Yaskawa INFORM job: DEMO_ROOF_SIDE_0625_3PAINT_4.JBI

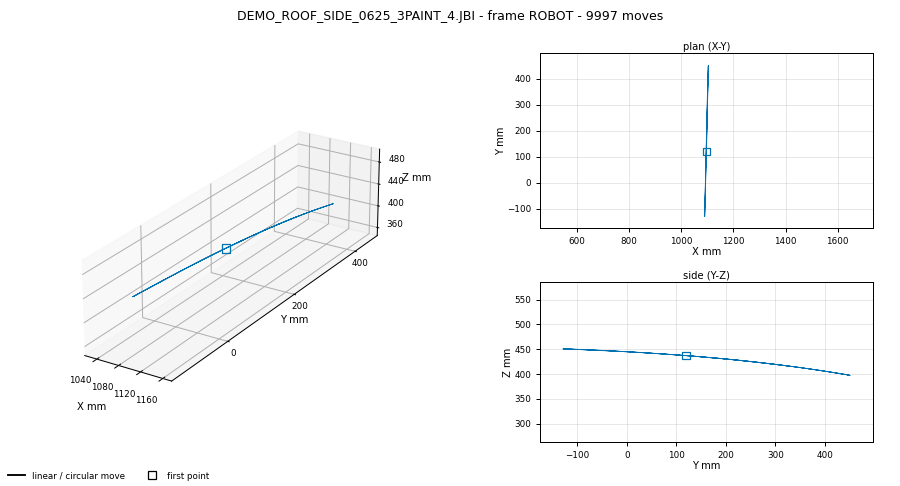
[picture p0: tool path of DEMO_ROOF_SIDE_0625_3PAINT_4.JBI in frame ROBOT, 9997 of 9997 moves have a stored position in this frame; points joined in program order, loops and branches not executed]
/JOB
//NAME DEMO_ROOF_SIDE_0625_3PAINT4
//POS
///NPOS 9997,0,0,0,0,0
///TOOL 0
///USER 0
///POSTYPE ROBOT
///RECTAN
///RCONF 1,0,0,0,0,0,0,0,0,0,0,0,0,0,0,0,0,0,0,0,0,0,0,0
C00000=1096.596,120.158,437.402,176.522,16.758,152.268
C00001=1096.602,120.407,437.382,176.524,16.758,152.268
C00002=1096.608,120.656,437.363,176.527,16.758,152.267
C00003=1096.614,120.905,437.344,176.530,16.759,152.267
C00004=1096.619,121.154,437.325,176.533,16.759,152.267
C00005=1096.625,121.404,437.306,176.536,16.760,152.266
C00006=1096.630,121.653,437.287,176.539,16.761,152.266
C00007=1096.636,121.902,437.267,176.541,16.761,152.265
C00008=1096.641,122.152,437.247,176.544,16.762,152.265
C00009=1096.646,122.400,437.228,176.546,16.761,152.264
C00010=1096.652,122.650,437.209,176.549,16.762,152.264
C00011=1096.658,122.899,437.189,176.552,16.763,152.263
C00012=1096.664,123.148,437.170,176.555,16.763,152.263
C00013=1096.669,123.397,437.150,176.558,16.764,152.262
C00014=1096.675,123.647,437.131,176.561,16.764,152.262
C00015=1096.681,123.896,437.111,176.563,16.765,152.262
C00016=1096.686,124.144,437.092,176.566,16.765,152.261
C00017=1096.692,124.394,437.073,176.569,16.766,152.261
C00018=1096.697,124.643,437.054,176.571,16.766,152.260
C00019=1096.703,124.892,437.034,176.575,16.766,152.260
C00020=1096.709,125.141,437.015,176.578,16.767,152.259
C00021=1096.715,125.391,436.995,176.580,16.767,152.259
C00022=1096.720,125.640,436.975,176.583,16.768,152.258
C00023=1096.726,125.889,436.955,176.585,16.768,152.258
C00024=1096.731,126.138,436.936,176.589,16.768,152.257
C00025=1096.737,126.387,436.917,176.592,16.769,152.257
C00026=1096.743,126.636,436.897,176.594,16.769,152.256
C00027=1096.749,126.885,436.877,176.597,16.770,152.256
C00028=1096.754,127.135,436.858,176.600,16.770,152.256
C00029=1096.760,127.383,436.838,176.602,16.770,152.255
C00030=1096.766,127.659,436.817,176.606,16.771,152.254
C00031=1096.773,127.934,436.795,176.609,16.771,152.254
C00032=1096.779,128.209,436.774,176.612,16.772,152.253
C00033=1096.785,128.484,436.751,176.615,16.772,152.253
C00034=1096.791,128.733,436.731,176.618,16.773,152.252
C00035=1096.796,128.982,436.712,176.621,16.773,152.252
C00036=1096.802,129.231,436.693,176.624,16.773,152.251
C00037=1096.808,129.480,436.673,176.627,16.774,152.251
C00038=1096.814,129.729,436.653,176.629,16.774,152.250
C00039=1096.819,129.979,436.634,176.632,16.774,152.250
C00040=1096.825,130.227,436.614,176.636,16.775,152.249
C00041=1096.830,130.477,436.594,176.638,16.775,152.249
C00042=1096.836,130.726,436.574,176.641,16.775,152.248
C00043=1096.842,130.975,436.555,176.644,16.776,152.248
C00044=1096.848,131.225,436.535,176.646,16.776,152.247
C00045=1096.854,131.474,436.514,176.649,16.777,152.247
C00046=1096.859,131.723,436.495,176.653,16.777,152.246
C00047=1096.865,131.972,436.475,176.655,16.777,152.246
C00048=1096.871,132.221,436.456,176.658,16.778,152.245
C00049=1096.876,132.470,436.435,176.661,16.778,152.245
C00050=1096.882,132.719,436.415,176.664,16.778,152.244
C00051=1096.888,132.969,436.396,176.667,16.778,152.244
C00052=1096.893,133.218,436.376,176.670,16.779,152.243
C00053=1096.899,133.467,436.356,176.672,16.779,152.243
C00054=1096.904,133.716,436.336,176.676,16.779,152.242
C00055=1096.910,133.965,436.316,176.679,16.780,152.242
C00056=1096.916,134.214,436.296,176.681,16.780,152.241
C00057=1096.921,134.464,436.276,176.684,16.781,152.241
C00058=1096.927,134.713,436.256,176.687,16.781,152.240
C00059=1096.932,134.962,436.235,176.690,16.781,152.240
C00060=1096.938,135.211,436.216,176.693,16.782,152.239
C00061=1096.944,135.460,436.196,176.696,16.782,152.239
C00062=1096.949,135.709,436.176,176.698,16.782,152.238
C00063=1096.955,135.958,436.156,176.701,16.783,152.238
C00064=1096.961,136.207,436.135,176.705,16.783,152.237
C00065=1096.966,136.456,436.116,176.707,16.783,152.237
C00066=1096.972,136.706,436.095,176.710,16.784,152.236
C00067=1096.978,136.954,436.075,176.713,16.784,152.236
C00068=1096.983,137.204,436.055,176.716,16.785,152.235
C00069=1096.989,137.452,436.035,176.719,16.785,152.235
C00070=1096.994,137.702,436.016,176.722,16.785,152.234
C00071=1097.000,137.951,435.995,176.725,16.785,152.234
C00072=1097.006,138.200,435.975,176.727,16.785,152.233
C00073=1097.012,138.450,435.954,176.731,16.786,152.233
C00074=1097.018,138.698,435.934,176.734,16.786,152.232
C00075=1097.023,138.947,435.914,176.736,16.786,152.232
C00076=1097.029,139.196,435.894,176.739,16.787,152.231
C00077=1097.034,139.446,435.874,176.743,16.787,152.231
C00078=1097.039,139.695,435.853,176.745,16.787,152.230
C00079=1097.045,139.944,435.833,176.748,16.788,152.230
C00080=1097.050,140.193,435.813,176.751,16.788,152.229
C00081=1097.056,140.442,435.793,176.755,16.788,152.228
C00082=1097.062,140.692,435.772,176.757,16.788,152.228
C00083=1097.068,140.941,435.752,176.760,16.789,152.227
C00084=1097.073,141.190,435.731,176.763,16.789,152.227
C00085=1097.079,141.439,435.711,176.766,16.789,152.226
C00086=1097.085,141.688,435.691,176.769,16.790,152.226
C00087=1097.090,141.937,435.670,176.772,16.790,152.225
C00088=1097.095,142.186,435.650,176.775,16.790,152.225
C00089=1097.101,142.435,435.630,176.778,16.790,152.224
C00090=1097.107,142.684,435.609,176.781,16.791,152.224
C00091=1097.112,142.934,435.588,176.784,16.791,152.223
C00092=1097.118,143.182,435.568,176.786,16.791,152.223
C00093=1097.124,143.432,435.548,176.790,16.792,152.222
C00094=1097.130,143.707,435.525,176.793,16.792,152.222
C00095=1097.136,143.981,435.503,176.797,16.792,152.221
C00096=1097.142,144.256,435.480,176.800,16.792,152.220
C00097=1097.149,144.530,435.458,176.803,16.793,152.220
C00098=1097.154,144.780,435.437,176.806,16.793,152.219
C00099=1097.160,145.029,435.416,176.809,16.793,152.219
C00100=1097.165,145.278,435.396,176.812,16.793,152.218
C00101=1097.171,145.527,435.376,176.815,16.794,152.218
C00102=1097.176,145.776,435.355,176.817,16.794,152.217
C00103=1097.182,146.025,435.333,176.821,16.794,152.216
C00104=1097.188,146.274,435.314,176.824,16.795,152.216
C00105=1097.194,146.523,435.293,176.827,16.795,152.215
C00106=1097.199,146.772,435.272,176.830,16.795,152.215
C00107=1097.205,147.022,435.251,176.833,16.795,152.214
C00108=1097.211,147.270,435.231,176.836,16.795,152.214
C00109=1097.216,147.519,435.210,176.839,16.795,152.213
C00110=1097.222,147.769,435.190,176.842,16.796,152.213
C00111=1097.227,148.018,435.169,176.845,16.796,152.212
C00112=1097.234,148.267,435.148,176.848,16.796,152.211
C00113=1097.239,148.516,435.128,176.851,16.796,152.211
C00114=1097.244,148.765,435.107,176.854,16.796,152.210
C00115=1097.250,149.015,435.086,176.857,16.797,152.210
C00116=1097.256,149.263,435.065,176.861,16.797,152.209
C00117=1097.261,149.512,435.044,176.863,16.797,152.209
C00118=1097.266,149.761,435.024,176.866,16.797,152.208
C00119=1097.273,150.010,435.003,176.870,16.798,152.207
C00120=1097.278,150.259,434.982,176.872,16.797,152.207
C00121=1097.284,150.509,434.962,176.875,16.798,152.206
C00122=1097.289,150.757,434.940,176.879,16.798,152.206
C00123=1097.295,151.007,434.919,176.882,16.799,152.205
C00124=1097.301,151.255,434.898,176.884,16.798,152.205
C00125=1097.306,151.505,434.878,176.888,16.799,152.204
C00126=1097.312,151.754,434.857,176.891,16.799,152.203
C00127=1097.317,152.003,434.835,176.894,16.799,152.203
C00128=1097.322,152.252,434.815,176.897,16.799,152.202
C00129=1097.329,152.501,434.793,176.900,16.800,152.202
C00130=1097.334,152.750,434.773,176.903,16.800,152.201
C00131=1097.339,152.999,434.751,176.906,16.800,152.201
C00132=1097.345,153.248,434.731,176.909,16.800,152.200
C00133=1097.351,153.497,434.710,176.912,16.801,152.200
C00134=1097.357,153.746,434.689,176.915,16.801,152.199
C00135=1097.362,153.995,434.669,176.918,16.800,152.198
C00136=1097.368,154.244,434.647,176.921,16.801,152.198
C00137=1097.374,154.493,434.626,176.925,16.801,152.197
C00138=1097.380,154.743,434.605,176.928,16.801,152.197
C00139=1097.385,154.991,434.584,176.930,16.801,152.196
C00140=1097.391,155.240,434.563,176.934,16.801,152.195
C00141=1097.397,155.489,434.541,176.937,16.802,152.195
C00142=1097.402,155.739,434.521,176.940,16.802,152.194
C00143=1097.407,155.987,434.499,176.943,16.802,152.194
C00144=1097.413,156.237,434.478,176.946,16.802,152.193
C00145=1097.418,156.486,434.457,176.949,16.802,152.192
C00146=1097.424,156.735,434.435,176.953,16.803,152.192
C00147=1097.430,156.984,434.415,176.955,16.802,152.191
C00148=1097.435,157.233,434.393,176.958,16.803,152.191
C00149=1097.441,157.482,434.372,176.962,16.803,152.190
C00150=1097.447,157.731,434.351,176.965,16.803,152.190
C00151=1097.452,157.979,434.330,176.968,16.803,152.189
C00152=1097.458,158.229,434.308,176.971,16.803,152.188
C00153=1097.463,158.478,434.287,176.974,16.804,152.188
C00154=1097.469,158.727,434.265,176.978,16.804,152.187
C00155=1097.475,158.976,434.244,176.980,16.803,152.187
C00156=1097.480,159.226,434.223,176.983,16.804,152.186
C00157=1097.486,159.474,434.202,176.987,16.804,152.185
C00158=1097.493,159.748,434.178,176.990,16.804,152.185
C00159=1097.499,160.023,434.155,176.994,16.804,152.184
C00160=1097.505,160.298,434.132,176.997,16.804,152.183
C00161=1097.510,160.572,434.107,177.001,16.804,152.183
C00162=1097.517,160.822,434.086,177.004,16.805,152.182
C00163=1097.522,161.070,434.064,177.007,16.805,152.181
C00164=1097.528,161.320,434.044,177.010,16.804,152.181
C00165=1097.533,161.568,434.022,177.013,16.805,152.180
C00166=1097.538,161.817,434.000,177.016,16.805,152.180
C00167=1097.544,162.066,433.979,177.020,16.805,152.179
C00168=1097.550,162.315,433.958,177.023,16.805,152.178
C00169=1097.555,162.564,433.935,177.026,16.805,152.178
C00170=1097.561,162.814,433.915,177.029,16.806,152.177
C00171=1097.566,163.063,433.893,177.032,16.806,152.177
C00172=1097.572,163.312,433.871,177.036,16.806,152.176
C00173=1097.577,163.560,433.850,177.038,16.806,152.175
C00174=1097.583,163.810,433.828,177.041,16.806,152.175
C00175=1097.588,164.058,433.806,177.045,16.806,152.174
C00176=1097.594,164.308,433.784,177.048,16.806,152.174
C00177=1097.599,164.556,433.763,177.051,16.807,152.173
C00178=1097.605,164.806,433.741,177.054,16.807,152.173
C00179=1097.610,165.054,433.719,177.057,16.807,152.172
C00180=1097.616,165.303,433.698,177.061,16.807,152.171
C00181=1097.621,165.552,433.676,177.064,16.807,152.171
C00182=1097.627,165.801,433.654,177.067,16.808,152.170
C00183=1097.632,166.050,433.632,177.070,16.807,152.169
C00184=1097.638,166.299,433.611,177.073,16.807,152.169
C00185=1097.643,166.548,433.589,177.076,16.808,152.168
C00186=1097.649,166.797,433.567,177.080,16.808,152.168
C00187=1097.654,167.046,433.545,177.083,16.808,152.167
C00188=1097.660,167.295,433.524,177.086,16.807,152.166
C00189=1097.665,167.544,433.502,177.089,16.808,152.166
C00190=1097.671,167.793,433.480,177.093,16.808,152.165
C00191=1097.676,168.042,433.458,177.096,16.808,152.164
C00192=1097.682,168.291,433.437,177.099,16.809,152.164
C00193=1097.687,168.540,433.415,177.102,16.808,152.163
C00194=1097.693,168.790,433.393,177.105,16.808,152.163
C00195=1097.698,169.038,433.371,177.109,16.809,152.162
C00196=1097.704,169.288,433.350,177.112,16.809,152.161
C00197=1097.709,169.536,433.327,177.115,16.808,152.161
C00198=1097.716,169.785,433.306,177.118,16.808,152.160
C00199=1097.721,170.034,433.283,177.121,16.809,152.159
C00200=1097.727,170.283,433.262,177.125,16.809,152.159
C00201=1097.732,170.532,433.240,177.128,16.809,152.158
C00202=1097.738,170.780,433.218,177.131,16.808,152.158
C00203=1097.743,171.030,433.196,177.134,16.809,152.157
C00204=1097.749,171.279,433.173,177.138,16.809,152.156
C00205=1097.754,171.528,433.152,177.141,16.809,152.156
C00206=1097.760,171.777,433.129,177.144,16.809,152.155
C00207=1097.766,172.026,433.108,177.148,16.809,152.154
C00208=1097.771,172.275,433.086,177.150,16.809,152.154
C00209=1097.777,172.524,433.064,177.154,16.809,152.153
C00210=1097.782,172.772,433.042,177.157,16.809,152.152
C00211=1097.788,173.022,433.019,177.161,16.810,152.152
C00212=1097.794,173.271,432.998,177.164,16.809,152.151
C00213=1097.799,173.519,432.975,177.167,16.809,152.150
C00214=1097.805,173.768,432.953,177.170,16.809,152.150
C00215=1097.811,174.018,432.931,177.174,16.809,152.149
C00216=1097.816,174.267,432.908,177.177,16.810,152.149
C00217=1097.822,174.515,432.887,177.180,16.809,152.148
C00218=1097.827,174.765,432.865,177.183,16.809,152.147
C00219=1097.833,175.014,432.842,177.186,16.809,152.147
C00220=1097.839,175.262,432.821,177.190,16.809,152.146
C00221=1097.844,175.511,432.798,177.193,16.809,152.145
C00222=1097.851,175.785,432.774,177.197,16.809,152.144
C00223=1097.857,176.060,432.749,177.201,16.809,152.144
C00224=1097.864,176.334,432.724,177.204,16.809,152.143
C00225=1097.869,176.608,432.700,177.208,16.809,152.142
C00226=1097.875,176.857,432.677,177.211,16.809,152.142
C00227=1097.881,177.106,432.656,177.214,16.809,152.141
C00228=1097.887,177.355,432.633,177.218,16.809,152.140
C00229=1097.892,177.604,432.611,177.222,16.809,152.140
C00230=1097.898,177.852,432.589,177.224,16.809,152.139
C00231=1097.903,178.102,432.566,177.228,16.809,152.138
C00232=1097.909,178.351,432.543,177.231,16.809,152.138
C00233=1097.914,178.600,432.521,177.234,16.809,152.137
C00234=1097.920,178.848,432.499,177.238,16.809,152.136
C00235=1097.926,179.097,432.476,177.241,16.809,152.136
C00236=1097.931,179.346,432.454,177.244,16.808,152.135
C00237=1097.938,179.595,432.432,177.248,16.808,152.134
C00238=1097.943,179.845,432.409,177.251,16.809,152.134
C00239=1097.949,180.093,432.386,177.254,16.809,152.133
C00240=1097.954,180.342,432.364,177.258,16.809,152.132
C00241=1097.960,180.591,432.342,177.262,16.809,152.131
C00242=1097.966,180.840,432.319,177.264,16.808,152.131
C00243=1097.972,181.089,432.296,177.268,16.808,152.130
C00244=1097.977,181.338,432.274,177.271,16.808,152.129
C00245=1097.984,181.587,432.252,177.275,16.808,152.129
C00246=1097.989,181.836,432.229,177.278,16.808,152.128
C00247=1097.994,182.084,432.207,177.282,16.808,152.127
C00248=1098.000,182.333,432.184,177.284,16.808,152.127
C00249=1098.006,182.582,432.162,177.288,16.808,152.126
C00250=1098.012,182.831,432.139,177.291,16.808,152.125
C00251=1098.018,183.080,432.117,177.295,16.808,152.125
C00252=1098.023,183.329,432.094,177.298,16.808,152.124
C00253=1098.029,183.578,432.071,177.302,16.808,152.123
C00254=1098.036,183.827,432.048,177.305,16.807,152.123
C00255=1098.041,184.076,432.025,177.308,16.807,152.122
C00256=1098.047,184.325,432.003,177.312,16.807,152.121
C00257=1098.052,184.573,431.981,177.315,16.807,152.120
C00258=1098.058,184.822,431.958,177.319,16.807,152.120
C00259=1098.063,185.071,431.935,177.322,16.807,152.119
C00260=1098.069,185.320,431.912,177.325,16.806,152.118
C00261=1098.075,185.569,431.889,177.328,16.807,152.118
C00262=1098.080,185.818,431.866,177.332,16.807,152.117
C00263=1098.086,186.067,431.844,177.335,16.807,152.116
C00264=1098.092,186.316,431.821,177.339,16.807,152.116
C00265=1098.097,186.564,431.798,177.342,16.807,152.115
C00266=1098.102,186.813,431.775,177.346,16.807,152.114
C00267=1098.108,187.062,431.752,177.349,16.807,152.114
C00268=1098.113,187.311,431.729,177.352,16.806,152.113
C00269=1098.119,187.560,431.706,177.355,16.806,152.112
C00270=1098.125,187.809,431.683,177.359,16.806,152.111
C00271=1098.130,188.058,431.660,177.362,16.807,152.111
C00272=1098.136,188.306,431.637,177.366,16.807,152.110
C00273=1098.141,188.555,431.614,177.369,16.807,152.109
C00274=1098.147,188.804,431.591,177.373,16.807,152.109
C00275=1098.152,189.053,431.568,177.376,16.806,152.108
C00276=1098.158,189.302,431.545,177.379,16.806,152.107
C00277=1098.163,189.551,431.522,177.383,16.806,152.107
C00278=1098.169,189.800,431.499,177.386,16.806,152.106
C00279=1098.175,190.049,431.476,177.389,16.806,152.105
C00280=1098.180,190.298,431.452,177.393,16.806,152.105
C00281=1098.186,190.547,431.429,177.397,16.806,152.104
C00282=1098.191,190.796,431.407,177.400,16.806,152.103
C00283=1098.197,191.045,431.384,177.404,16.806,152.102
C00284=1098.203,191.294,431.361,177.406,16.805,152.102
C00285=1098.208,191.542,431.336,177.410,16.805,152.101
C00286=1098.214,191.816,431.311,177.413,16.805,152.100
C00287=1098.220,192.090,431.286,177.418,16.805,152.099
C00288=1098.226,192.363,431.260,177.422,16.805,152.099
C00289=1098.232,192.637,431.235,177.425,16.805,152.098
C00290=1098.238,192.886,431.212,177.429,16.805,152.097
C00291=1098.243,193.135,431.189,177.433,16.805,152.096
C00292=1098.249,193.384,431.166,177.436,16.805,152.096
C00293=1098.255,193.632,431.142,177.440,16.805,152.095
C00294=1098.261,193.881,431.119,177.442,16.804,152.094
C00295=1098.266,194.130,431.095,177.446,16.804,152.094
C00296=1098.271,194.379,431.072,177.449,16.804,152.093
C00297=1098.277,194.628,431.049,177.453,16.804,152.092
C00298=1098.283,194.877,431.026,177.456,16.804,152.091
C00299=1098.289,195.126,431.002,177.460,16.804,152.091
C00300=1098.295,195.375,430.978,177.464,16.804,152.090
C00301=1098.301,195.624,430.955,177.467,16.804,152.089
C00302=1098.306,195.873,430.932,177.471,16.804,152.089
C00303=1098.312,196.121,430.908,177.473,16.803,152.088
C00304=1098.317,196.370,430.885,177.477,16.803,152.087
C00305=1098.322,196.619,430.862,177.480,16.803,152.087
C00306=1098.328,196.867,430.838,177.484,16.803,152.086
C00307=1098.334,197.116,430.815,177.487,16.803,152.085
C00308=1098.339,197.366,430.792,177.491,16.803,152.084
C00309=1098.345,197.614,430.768,177.495,16.803,152.083
C00310=1098.351,197.863,430.745,177.498,16.803,152.083
C00311=1098.357,198.112,430.720,177.502,16.803,152.082
C00312=1098.362,198.361,430.697,177.505,16.803,152.081
C00313=1098.368,198.609,430.674,177.508,16.802,152.081
C00314=1098.373,198.858,430.650,177.512,16.802,152.080
C00315=1098.380,199.107,430.626,177.516,16.802,152.079
C00316=1098.384,199.356,430.603,177.519,16.802,152.078
C00317=1098.391,199.605,430.579,177.523,16.802,152.078
C00318=1098.397,199.854,430.556,177.526,16.802,152.077
C00319=1098.402,200.102,430.532,177.530,16.802,152.076
C00320=1098.408,200.351,430.509,177.533,16.801,152.075
C00321=1098.414,200.600,430.485,177.537,16.801,152.075
C00322=1098.419,200.849,430.462,177.541,16.801,152.074
C00323=1098.426,201.098,430.438,177.544,16.801,152.073
C00324=1098.431,201.347,430.414,177.547,16.800,152.072
C00325=1098.437,201.595,430.390,177.551,16.800,152.072
C00326=1098.442,201.844,430.366,177.554,16.800,152.071
C00327=1098.448,202.093,430.343,177.558,16.800,152.070
C00328=1098.454,202.342,430.319,177.562,16.800,152.069
C00329=1098.460,202.590,430.295,177.565,16.800,152.069
C00330=1098.465,202.839,430.272,177.569,16.799,152.068
C00331=1098.471,203.088,430.248,177.572,16.799,152.067
C00332=1098.476,203.337,430.223,177.576,16.799,152.067
C00333=1098.482,203.586,430.200,177.580,16.799,152.066
C00334=1098.488,203.835,430.176,177.583,16.799,152.065
C00335=1098.494,204.083,430.152,177.587,16.799,152.064
C00336=1098.499,204.332,430.129,177.590,16.799,152.064
C00337=1098.504,204.581,430.104,177.594,16.799,152.063
C00338=1098.510,204.830,430.080,177.597,16.798,152.062
C00339=1098.516,205.078,430.056,177.600,16.798,152.061
C00340=1098.521,205.327,430.033,177.604,16.798,152.061
C00341=1098.527,205.576,430.009,177.607,16.798,152.060
C00342=1098.533,205.825,429.984,177.611,16.797,152.059
C00343=1098.538,206.074,429.960,177.615,16.797,152.058
C00344=1098.544,206.322,429.937,177.618,16.797,152.058
C00345=1098.549,206.571,429.913,177.622,16.797,152.057
C00346=1098.555,206.820,429.888,177.626,16.797,152.056
C00347=1098.561,207.069,429.865,177.629,16.797,152.055
C00348=1098.566,207.317,429.840,177.633,16.797,152.055
C00349=1098.572,207.566,429.816,177.636,16.797,152.054
C00350=1098.595,208.576,429.718,177.680,16.812,152.049
C00351=1098.603,208.947,429.682,177.685,16.813,152.048
C00352=1098.611,209.317,429.646,177.690,16.814,152.047
C00353=1098.620,209.688,429.610,177.695,16.815,152.046
C00354=1098.629,210.058,429.573,177.699,16.816,152.045
C00355=1098.634,210.306,429.549,177.703,16.817,152.045
C00356=1098.640,210.555,429.524,177.707,16.817,152.044
C00357=1098.645,210.804,429.500,177.710,16.818,152.044
C00358=1098.651,211.053,429.476,177.713,16.818,152.043
C00359=1098.657,211.302,429.451,177.717,16.820,152.043
C00360=1098.662,211.550,429.427,177.720,16.820,152.042
C00361=1098.668,211.799,429.401,177.723,16.821,152.042
C00362=1098.673,212.048,429.377,177.726,16.821,152.041
C00363=1098.679,212.296,429.353,177.730,16.822,152.041
C00364=1098.685,212.546,429.328,177.734,16.823,152.040
C00365=1098.690,212.794,429.304,177.737,16.824,152.040
C00366=1098.696,213.043,429.279,177.740,16.824,152.039
C00367=1098.701,213.291,429.254,177.744,16.825,152.039
C00368=1098.707,213.541,429.230,177.747,16.826,152.038
C00369=1098.713,213.789,429.205,177.750,16.826,152.038
C00370=1098.718,214.037,429.180,177.753,16.827,152.037
C00371=1098.724,214.287,429.156,177.757,16.828,152.037
C00372=1098.729,214.535,429.132,177.761,16.829,152.036
C00373=1098.736,214.784,429.106,177.764,16.830,152.036
C00374=1098.741,215.032,429.082,177.768,16.831,152.035
C00375=1098.747,215.282,429.057,177.771,16.831,152.034
C00376=1098.752,215.530,429.032,177.774,16.832,152.034
C00377=1098.757,215.779,429.008,177.777,16.832,152.034
C00378=1098.763,216.028,428.983,177.781,16.834,152.033
C00379=1098.768,216.276,428.958,177.784,16.834,152.032
C00380=1098.774,216.525,428.933,177.787,16.835,152.032
C00381=1098.780,216.773,428.908,177.790,16.835,152.032
C00382=1098.786,217.022,428.884,177.794,16.836,152.031
C00383=1098.791,217.271,428.858,177.798,16.837,152.030
C00384=1098.797,217.520,428.834,177.801,16.838,152.030
C00385=1098.802,217.768,428.809,177.805,16.839,152.029
C00386=1098.808,218.017,428.784,177.808,16.839,152.029
C00387=1098.814,218.265,428.759,177.811,16.840,152.028
C00388=1098.819,218.515,428.734,177.815,16.841,152.028
C00389=1098.825,218.763,428.708,177.818,16.842,152.027
C00390=1098.830,219.012,428.684,177.821,16.842,152.027
C00391=1098.837,219.261,428.659,177.825,16.843,152.026
C00392=1098.842,219.509,428.635,177.828,16.844,152.026
C00393=1098.847,219.758,428.609,177.832,16.845,152.025
C00394=1098.853,220.007,428.584,177.835,16.845,152.025
C00395=1098.859,220.256,428.559,177.839,16.846,152.024
C00396=1098.865,220.504,428.534,177.842,16.847,152.024
C00397=1098.870,220.753,428.509,177.845,16.848,152.023
C00398=1098.876,221.002,428.484,177.848,16.848,152.023
C00399=1098.881,221.250,428.459,177.852,16.849,152.022
C00400=1098.887,221.499,428.434,177.856,16.850,152.022
C00401=1098.893,221.748,428.408,177.858,16.851,152.021
C00402=1098.898,221.996,428.383,177.863,16.852,152.021
C00403=1098.907,222.371,428.346,177.868,16.853,152.020
C00404=1098.915,222.745,428.308,177.873,16.854,152.019
C00405=1098.923,223.119,428.269,177.878,16.855,152.018
C00406=1098.932,223.494,428.231,177.883,16.857,152.018
C00407=1098.937,223.742,428.206,177.886,16.857,152.017
C00408=1098.943,223.991,428.181,177.889,16.857,152.017
C00409=1098.949,224.240,428.156,177.893,16.859,152.016
C00410=1098.954,224.488,428.130,177.896,16.859,152.016
C00411=1098.960,224.737,428.105,177.900,16.860,152.015
C00412=1098.966,224.986,428.079,177.903,16.861,152.015
C00413=1098.971,225.234,428.054,177.907,16.862,152.014
C00414=1098.977,225.484,428.029,177.910,16.862,152.014
C00415=1098.982,225.731,428.004,177.914,16.864,152.013
C00416=1098.988,225.980,427.978,177.917,16.864,152.013
C00417=1098.994,226.229,427.953,177.920,16.865,152.012
C00418=1098.999,226.478,427.927,177.924,16.866,152.012
C00419=1099.005,226.726,427.902,177.927,16.867,152.011
C00420=1099.010,226.975,427.876,177.930,16.867,152.011
C00421=1099.017,227.224,427.850,177.934,16.869,152.010
C00422=1099.022,227.472,427.825,177.937,16.869,152.010
C00423=1099.028,227.721,427.800,177.940,16.870,152.009
C00424=1099.033,227.970,427.774,177.944,16.871,152.009
C00425=1099.039,228.218,427.748,177.947,16.872,152.008
C00426=1099.044,228.467,427.723,177.951,16.873,152.008
C00427=1099.051,228.715,427.697,177.955,16.873,152.007
C00428=1099.056,228.964,427.671,177.958,16.874,152.007
C00429=1099.062,229.213,427.646,177.962,16.875,152.006
C00430=1099.067,229.461,427.621,177.965,16.876,152.006
C00431=1099.073,229.710,427.595,177.968,16.876,152.005
C00432=1099.079,229.959,427.569,177.972,16.878,152.005
C00433=1099.084,230.208,427.543,177.975,16.878,152.004
C00434=1099.090,230.456,427.518,177.978,16.879,152.004
C00435=1099.095,230.705,427.492,177.982,16.880,152.003
C00436=1099.101,230.954,427.467,177.985,16.881,152.003
C00437=1099.107,231.202,427.440,177.989,16.882,152.002
C00438=1099.112,231.450,427.415,177.992,16.883,152.002
C00439=1099.118,231.699,427.389,177.995,16.883,152.001
C00440=1099.124,231.948,427.364,177.999,16.885,152.001
C00441=1099.129,232.197,427.338,178.002,16.885,152.000
C00442=1099.135,232.445,427.311,178.006,16.886,152.000
C00443=1099.141,232.693,427.286,178.009,16.887,151.999
C00444=1099.146,232.942,427.260,178.013,16.888,151.999
C00445=1099.152,233.191,427.234,178.017,16.889,151.998
C00446=1099.157,233.440,427.208,178.020,16.890,151.998
C00447=1099.164,233.688,427.182,178.023,16.890,151.997
C00448=1099.168,233.936,427.157,178.027,16.891,151.997
C00449=1099.174,234.185,427.131,178.030,16.892,151.996
C00450=1099.180,234.434,427.104,178.034,16.893,151.996
C00451=1099.185,234.683,427.078,178.037,16.894,151.995
C00452=1099.191,234.931,427.053,178.040,16.895,151.995
C00453=1099.197,235.180,427.026,178.044,16.896,151.994
C00454=1099.202,235.428,427.001,178.047,16.897,151.994
C00455=1099.211,235.794,426.962,178.052,16.898,151.993
C00456=1099.218,236.160,426.923,178.057,16.899,151.992
C00457=1099.227,236.526,426.885,178.062,16.901,151.992
C00458=1099.235,236.891,426.847,178.067,16.902,151.991
C00459=1099.241,237.140,426.821,178.071,16.903,151.991
C00460=1099.246,237.389,426.794,178.074,16.904,151.990
C00461=1099.252,237.638,426.768,178.077,16.905,151.990
C00462=1099.258,237.886,426.742,178.081,16.906,151.989
C00463=1099.263,238.134,426.716,178.084,16.907,151.989
C00464=1099.269,238.382,426.690,178.088,16.908,151.988
C00465=1099.275,238.631,426.664,178.091,16.909,151.988
C00466=1099.280,238.880,426.637,178.094,16.909,151.987
C00467=1099.286,239.129,426.611,178.098,16.911,151.987
C00468=1099.292,239.377,426.585,178.101,16.911,151.986
C00469=1099.297,239.626,426.559,178.105,16.913,151.986
C00470=1099.303,239.874,426.532,178.109,16.913,151.985
C00471=1099.309,240.123,426.506,178.112,16.915,151.985
C00472=1099.314,240.372,426.480,178.116,16.915,151.984
C00473=1099.320,240.620,426.453,178.119,16.916,151.984
C00474=1099.325,240.869,426.427,178.123,16.917,151.983
C00475=1099.331,241.118,426.400,178.126,16.918,151.983
C00476=1099.337,241.366,426.374,178.130,16.919,151.982
C00477=1099.342,241.615,426.348,178.133,16.920,151.982
C00478=1099.348,241.863,426.321,178.136,16.921,151.982
C00479=1099.354,242.112,426.295,178.140,16.922,151.981
C00480=1099.360,242.360,426.268,178.143,16.923,151.981
C00481=1099.365,242.609,426.242,178.147,16.924,151.980
C00482=1099.371,242.857,426.215,178.150,16.924,151.980
C00483=1099.377,243.106,426.189,178.154,16.926,151.979
C00484=1099.382,243.354,426.162,178.157,16.926,151.979
C00485=1099.387,243.603,426.135,178.161,16.928,151.978
C00486=1099.393,243.852,426.109,178.164,16.928,151.978
C00487=1099.399,244.100,426.082,178.168,16.930,151.977
C00488=1099.405,244.348,426.056,178.171,16.930,151.977
C00489=1099.410,244.597,426.029,178.175,16.932,151.976
C00490=1099.416,244.846,426.003,178.178,16.932,151.976
C00491=1099.421,245.094,425.976,178.181,16.934,151.975
C00492=1099.427,245.343,425.949,178.185,16.934,151.975
C00493=1099.432,245.591,425.922,178.188,16.935,151.975
C00494=1099.438,245.839,425.896,178.192,16.937,151.974
C00495=1099.444,246.088,425.869,178.195,16.937,151.974
C00496=1099.449,246.336,425.842,178.199,16.939,151.973
C00497=1099.455,246.585,425.815,178.202,16.939,151.973
C00498=1099.460,246.833,425.789,178.206,16.941,151.972
C00499=1099.466,247.082,425.762,178.209,16.942,151.972
C00500=1099.472,247.331,425.734,178.213,16.943,151.971
C00501=1099.478,247.579,425.708,178.215,16.944,151.971
C00502=1099.483,247.828,425.681,178.219,16.945,151.970
C00503=1099.488,248.076,425.654,178.222,16.946,151.970
C00504=1099.494,248.325,425.627,178.226,16.947,151.970
C00505=1099.499,248.573,425.600,178.229,16.948,151.969
C00506=1099.505,248.822,425.573,178.233,16.949,151.969
C00507=1099.513,249.180,425.535,178.238,16.951,151.968
C00508=1099.521,249.540,425.496,178.243,16.952,151.967
C00509=1099.529,249.899,425.456,178.248,16.954,151.967
C00510=1099.537,250.257,425.418,178.253,16.955,151.966
C00511=1099.542,250.506,425.391,178.256,16.956,151.966
C00512=1099.548,250.754,425.364,178.260,16.957,151.965
C00513=1099.553,251.003,425.336,178.263,16.958,151.965
C00514=1099.560,251.252,425.309,178.267,16.960,151.964
C00515=1099.565,251.500,425.282,178.270,16.960,151.964
C00516=1099.570,251.749,425.255,178.273,16.962,151.963
C00517=1099.576,251.997,425.229,178.277,16.962,151.963
C00518=1099.582,252.245,425.201,178.280,16.964,151.963
C00519=1099.587,252.493,425.174,178.284,16.965,151.962
C00520=1099.593,252.743,425.146,178.287,16.966,151.962
C00521=1099.599,252.991,425.120,178.291,16.968,151.961
C00522=1099.604,253.239,425.092,178.294,16.968,151.961
C00523=1099.610,253.488,425.065,178.298,16.970,151.960
C00524=1099.615,253.736,425.038,178.301,16.971,151.960
C00525=1099.621,253.985,425.011,178.305,16.972,151.959
C00526=1099.627,254.233,424.983,178.308,16.973,151.959
C00527=1099.632,254.482,424.956,178.312,16.974,151.959
C00528=1099.638,254.730,424.928,178.315,16.975,151.958
C00529=1099.643,254.978,424.902,178.319,16.976,151.958
C00530=1099.649,255.227,424.874,178.322,16.977,151.957
C00531=1099.654,255.476,424.846,178.326,16.978,151.957
C00532=1099.660,255.724,424.819,178.329,16.979,151.956
C00533=1099.666,255.972,424.791,178.333,16.980,151.956
C00534=1099.672,256.221,424.764,178.335,16.981,151.955
C00535=1099.677,256.470,424.737,178.339,16.982,151.955
C00536=1099.683,256.717,424.710,178.342,16.983,151.955
C00537=1099.688,256.966,424.683,178.346,16.985,151.954
C00538=1099.694,257.215,424.654,178.350,16.986,151.954
C00539=1099.700,257.463,424.628,178.353,16.987,151.953
C00540=1099.705,257.711,424.600,178.357,16.989,151.953
C00541=1099.712,257.960,424.573,178.360,16.989,151.952
C00542=1099.717,258.208,424.545,178.364,16.991,151.952
C00543=1099.722,258.456,424.517,178.367,16.991,151.951
C00544=1099.729,258.705,424.490,178.371,16.993,151.951
C00545=1099.734,258.954,424.462,178.374,16.994,151.951
C00546=1099.740,259.202,424.435,178.378,16.995,151.950
C00547=1099.746,259.451,424.407,178.381,16.996,151.950
C00548=1099.751,259.699,424.379,178.384,16.997,151.949
C00549=1099.757,259.947,424.352,178.388,16.998,151.949
C00550=1099.763,260.196,424.324,178.391,16.999,151.948
C00551=1099.768,260.444,424.296,178.395,17.001,151.948
C00552=1099.774,260.692,424.269,178.398,17.001,151.948
C00553=1099.780,260.941,424.241,178.402,17.003,151.947
C00554=1099.785,261.189,424.213,178.405,17.004,151.947
C00555=1099.791,261.438,424.186,178.409,17.005,151.946
C00556=1099.797,261.686,424.158,178.412,17.006,151.946
C00557=1099.802,261.934,424.130,178.416,17.007,151.945
C00558=1099.808,262.183,424.102,178.420,17.009,151.945
C00559=1099.816,262.539,424.062,178.425,17.010,151.944
C00560=1099.825,262.895,424.022,178.429,17.012,151.944
C00561=1099.833,263.251,423.982,178.434,17.014,151.943
C00562=1099.841,263.607,423.943,178.439,17.015,151.942
C00563=1099.846,263.856,423.915,178.443,17.016,151.942
C00564=1099.853,264.104,423.887,178.446,17.017,151.942
C00565=1099.858,264.352,423.859,178.450,17.018,151.941
C00566=1099.864,264.601,423.831,178.453,17.019,151.941
C00567=1099.870,264.849,423.803,178.457,17.021,151.940
C00568=1099.875,265.097,423.775,178.460,17.022,151.940
C00569=1099.881,265.346,423.747,178.464,17.023,151.940
C00570=1099.886,265.594,423.719,178.467,17.025,151.939
C00571=1099.892,265.842,423.690,178.470,17.026,151.939
C00572=1099.897,266.091,423.663,178.474,17.027,151.938
C00573=1099.904,266.340,423.635,178.477,17.028,151.938
C00574=1099.909,266.588,423.607,178.481,17.029,151.937
C00575=1099.915,266.836,423.579,178.485,17.031,151.937
C00576=1099.921,267.084,423.551,178.488,17.032,151.937
C00577=1099.926,267.332,423.522,178.491,17.033,151.936
C00578=1099.932,267.581,423.494,178.495,17.035,151.936
C00579=1099.938,267.829,423.466,178.498,17.036,151.936
C00580=1099.944,268.077,423.438,178.502,17.037,151.935
C00581=1099.949,268.325,423.410,178.505,17.038,151.935
C00582=1099.955,268.574,423.381,178.509,17.040,151.934
C00583=1099.960,268.822,423.353,178.512,17.041,151.934
C00584=1099.966,269.071,423.325,178.515,17.042,151.934
C00585=1099.971,269.319,423.297,178.519,17.043,151.933
C00586=1099.977,269.567,423.268,178.522,17.044,151.933
C00587=1099.982,269.816,423.240,178.526,17.046,151.932
C00588=1099.988,270.064,423.211,178.530,17.047,151.932
C00589=1099.994,270.312,423.183,178.533,17.048,151.932
C00590=1099.999,270.561,423.155,178.536,17.050,151.931
C00591=1100.006,270.809,423.126,178.540,17.051,151.931
C00592=1100.011,271.057,423.098,178.543,17.052,151.930
C00593=1100.017,271.306,423.070,178.547,17.054,151.930
C00594=1100.022,271.554,423.042,178.550,17.055,151.930
C00595=1100.028,271.803,423.012,178.554,17.056,151.929
C00596=1100.033,272.051,422.984,178.557,17.058,151.929
C00597=1100.039,272.299,422.956,178.560,17.059,151.928
C00598=1100.045,272.547,422.927,178.564,17.060,151.928
C00599=1100.051,272.795,422.899,178.568,17.062,151.928
C00600=1100.057,273.044,422.870,178.571,17.063,151.927
C00601=1100.062,273.292,422.841,178.574,17.064,151.927
C00602=1100.068,273.541,422.813,178.578,17.066,151.927
C00603=1100.073,273.789,422.785,178.581,17.067,151.926
C00604=1100.079,274.037,422.756,178.585,17.068,151.926
C00605=1100.084,274.286,422.727,178.588,17.070,151.925
C00606=1100.090,274.533,422.698,178.591,17.071,151.925
C00607=1100.096,274.782,422.670,178.595,17.073,151.925
C00608=1100.102,275.030,422.641,178.599,17.074,151.924
C00609=1100.107,275.279,422.612,178.602,17.075,151.924
C00610=1100.113,275.527,422.584,178.605,17.077,151.924
C00611=1100.121,275.885,422.542,178.610,17.078,151.923
C00612=1100.129,276.245,422.500,178.615,17.080,151.923
C00613=1100.137,276.603,422.459,178.621,17.083,151.922
C00614=1100.145,276.962,422.417,178.625,17.084,151.921
C00615=1100.151,277.210,422.389,178.629,17.086,151.921
C00616=1100.156,277.459,422.360,178.632,17.087,151.921
C00617=1100.163,277.707,422.331,178.636,17.088,151.920
C00618=1100.168,277.955,422.303,178.640,17.090,151.920
C00619=1100.173,278.203,422.273,178.642,17.091,151.920
C00620=1100.180,278.451,422.244,178.646,17.093,151.919
C00621=1100.184,278.700,422.216,178.650,17.094,151.919
C00622=1100.191,278.948,422.186,178.654,17.096,151.918
C00623=1100.196,279.196,422.157,178.656,17.097,151.918
C00624=1100.201,279.444,422.129,178.660,17.099,151.918
C00625=1100.208,279.693,422.100,178.664,17.100,151.918
C00626=1100.213,279.941,422.070,178.667,17.101,151.917
C00627=1100.219,280.190,422.042,178.670,17.103,151.917
C00628=1100.224,280.438,422.013,178.674,17.104,151.916
C00629=1100.230,280.686,421.984,178.677,17.105,151.916
C00630=1100.236,280.934,421.954,178.681,17.107,151.916
C00631=1100.241,281.182,421.925,178.684,17.109,151.915
C00632=1100.247,281.431,421.896,178.687,17.110,151.915
C00633=1100.253,281.679,421.867,178.691,17.111,151.915
C00634=1100.258,281.927,421.838,178.694,17.113,151.914
C00635=1100.264,282.175,421.809,178.698,17.115,151.914
C00636=1100.270,282.423,421.779,178.701,17.116,151.914
C00637=1100.275,282.671,421.750,178.705,17.117,151.913
C00638=1100.281,282.920,421.721,178.708,17.119,151.913
C00639=1100.286,283.168,421.692,178.711,17.120,151.913
C00640=1100.292,283.416,421.663,178.715,17.122,151.912
C00641=1100.298,283.665,421.633,178.719,17.123,151.912
C00642=1100.303,283.913,421.604,178.722,17.125,151.912
C00643=1100.309,284.160,421.575,178.725,17.126,151.911
C00644=1100.314,284.409,421.546,178.729,17.128,151.911
C00645=1100.320,284.657,421.516,178.732,17.130,151.911
C00646=1100.326,284.905,421.487,178.736,17.131,151.910
C00647=1100.332,285.154,421.457,178.739,17.133,151.910
C00648=1100.337,285.402,421.428,178.743,17.134,151.910
C00649=1100.343,285.650,421.399,178.746,17.136,151.909
C00650=1100.348,285.898,421.369,178.749,17.137,151.909
C00651=1100.354,286.147,421.340,178.753,17.139,151.909
C00652=1100.360,286.394,421.310,178.756,17.140,151.908
C00653=1100.365,286.642,421.281,178.760,17.142,151.908
C00654=1100.371,286.890,421.251,178.763,17.143,151.908
C00655=1100.377,287.138,421.222,178.766,17.145,151.907
C00656=1100.383,287.387,421.192,178.770,17.147,151.907
C00657=1100.388,287.635,421.163,178.774,17.148,151.907
C00658=1100.394,287.884,421.133,178.777,17.149,151.906
C00659=1100.400,288.131,421.103,178.780,17.151,151.906
C00660=1100.405,288.379,421.074,178.784,17.153,151.906
C00661=1100.411,288.627,421.044,178.788,17.154,151.905
C00662=1100.416,288.876,421.015,178.790,17.156,151.905
C00663=1100.425,289.245,420.971,178.796,17.158,151.905
C00664=1100.433,289.613,420.927,178.801,17.161,151.904
C00665=1100.442,289.981,420.883,178.806,17.163,151.904
C00666=1100.450,290.348,420.838,178.811,17.166,151.903
C00667=1100.456,290.596,420.809,178.815,17.167,151.903
C00668=1100.462,290.845,420.779,178.818,17.168,151.903
C00669=1100.467,291.093,420.749,178.821,17.170,151.902
C00670=1100.473,291.341,420.719,178.825,17.172,151.902
C00671=1100.478,291.590,420.690,178.828,17.174,151.902
C00672=1100.484,291.837,420.659,178.832,17.175,151.902
C00673=1100.490,292.086,420.630,178.835,17.177,151.901
C00674=1100.496,292.334,420.599,178.838,17.178,151.901
C00675=1100.501,292.582,420.570,178.842,17.180,151.901
C00676=1100.507,292.831,420.540,178.846,17.182,151.900
C00677=1100.512,293.078,420.510,178.849,17.183,151.900
C00678=1100.518,293.327,420.480,178.852,17.185,151.900
C00679=1100.523,293.574,420.450,178.856,17.187,151.899
C00680=1100.529,293.822,420.421,178.859,17.189,151.899
C00681=1100.535,294.070,420.391,178.863,17.190,151.899
C00682=1100.541,294.318,420.361,178.865,17.192,151.899
C00683=1100.547,294.566,420.331,178.869,17.193,151.898
C00684=1100.552,294.814,420.300,178.873,17.195,151.898
C00685=1100.557,295.063,420.270,178.876,17.197,151.898
C00686=1100.563,295.310,420.240,178.880,17.199,151.898
C00687=1100.569,295.559,420.210,178.883,17.200,151.897
C00688=1100.574,295.807,420.180,178.886,17.202,151.897
C00689=1100.580,296.055,420.149,178.890,17.203,151.897
C00690=1100.586,296.303,420.120,178.893,17.205,151.896
C00691=1100.591,296.551,420.089,178.897,17.207,151.896
C00692=1100.597,296.799,420.059,178.900,17.209,151.896
C00693=1100.603,297.048,420.029,178.904,17.211,151.896
C00694=1100.609,297.296,419.999,178.907,17.212,151.895
C00695=1100.615,297.543,419.968,178.910,17.214,151.895
C00696=1100.621,297.792,419.939,178.914,17.216,151.895
C00697=1100.626,298.040,419.908,178.917,17.218,151.895
C00698=1100.631,298.288,419.877,178.921,17.220,151.894
C00699=1100.637,298.536,419.847,178.924,17.221,151.894
C00700=1100.643,298.784,419.818,178.927,17.223,151.894
C00701=1100.648,299.032,419.787,178.931,17.225,151.894
C00702=1100.654,299.280,419.756,178.934,17.227,151.893
C00703=1100.659,299.528,419.726,178.938,17.228,151.893
C00704=1100.665,299.776,419.696,178.941,17.230,151.893
C00705=1100.670,300.024,419.665,178.945,17.233,151.893
C00706=1100.676,300.272,419.635,178.948,17.235,151.892
C00707=1100.682,300.520,419.605,178.951,17.236,151.892
C00708=1100.687,300.768,419.574,178.954,17.238,151.892
C00709=1100.693,301.016,419.543,178.958,17.240,151.892
C00710=1100.698,301.264,419.513,178.961,17.242,151.891
C00711=1100.704,301.512,419.482,178.965,17.244,151.891
C00712=1100.709,301.760,419.452,178.968,17.246,151.891
C00713=1100.714,302.008,419.421,178.972,17.247,151.891
C00714=1100.720,302.256,419.390,178.975,17.249,151.891
C00715=1100.730,302.638,419.343,178.980,17.253,151.890
C00716=1100.737,303.020,419.296,178.985,17.255,151.890
C00717=1100.747,303.403,419.248,178.991,17.258,151.890
C00718=1100.755,303.784,419.201,178.996,17.261,151.889
C00719=1100.760,304.032,419.170,178.999,17.263,151.889
C00720=1100.766,304.280,419.140,179.003,17.265,151.889
C00721=1100.772,304.529,419.109,179.005,17.267,151.889
C00722=1100.778,304.777,419.078,179.009,17.269,151.888
C00723=1100.783,305.024,419.048,179.012,17.271,151.888
C00724=1100.789,305.273,419.017,179.016,17.273,151.888
C00725=1100.795,305.520,418.986,179.019,17.274,151.888
C00726=1100.800,305.768,418.955,179.023,17.276,151.887
C00727=1100.806,306.016,418.924,179.026,17.278,151.887
C00728=1100.811,306.265,418.893,179.030,17.280,151.887
C00729=1100.817,306.512,418.863,179.033,17.282,151.887
C00730=1100.822,306.760,418.831,179.037,17.284,151.887
C00731=1100.828,307.008,418.801,179.040,17.286,151.886
C00732=1100.834,307.257,418.770,179.043,17.288,151.886
C00733=1100.840,307.504,418.739,179.046,17.290,151.886
C00734=1100.845,307.752,418.708,179.050,17.292,151.886
C00735=1100.851,308.000,418.677,179.053,17.294,151.886
C00736=1100.857,308.249,418.646,179.056,17.296,151.885
C00737=1100.863,308.496,418.615,179.060,17.298,151.885
C00738=1100.868,308.744,418.584,179.063,17.300,151.885
C00739=1100.875,308.992,418.553,179.067,17.302,151.885
C00740=1100.880,309.240,418.522,179.070,17.304,151.885
C00741=1100.885,309.488,418.491,179.074,17.306,151.884
C00742=1100.891,309.736,418.459,179.077,17.308,151.884
C00743=1100.897,309.984,418.428,179.080,17.310,151.884
C00744=1100.903,310.231,418.397,179.084,17.312,151.884
C00745=1100.908,310.480,418.366,179.087,17.314,151.884
C00746=1100.914,310.728,418.336,179.091,17.316,151.883
C00747=1100.920,310.975,418.304,179.094,17.318,151.883
C00748=1100.925,311.224,418.273,179.097,17.320,151.883
C00749=1100.931,311.471,418.242,179.100,17.322,151.883
C00750=1100.936,311.720,418.211,179.104,17.324,151.883
C00751=1100.943,311.968,418.179,179.107,17.326,151.882
C00752=1100.949,312.215,418.148,179.110,17.328,151.882
C00753=1100.954,312.464,418.116,179.114,17.330,151.882
C00754=1100.960,312.711,418.085,179.117,17.332,151.882
C00755=1100.965,312.959,418.054,179.120,17.334,151.882
C00756=1100.971,313.207,418.022,179.124,17.336,151.882
C00757=1100.978,313.455,417.991,179.127,17.338,151.881
C00758=1100.983,313.703,417.960,179.131,17.340,151.881
C00759=1100.989,313.951,417.928,179.134,17.342,151.881
C00760=1100.995,314.199,417.897,179.138,17.345,151.881
C00761=1101.000,314.447,417.866,179.141,17.347,151.881
C00762=1101.006,314.695,417.834,179.144,17.349,151.881
C00763=1101.012,314.943,417.802,179.148,17.351,151.880
C00764=1101.018,315.191,417.772,179.151,17.353,151.880
C00765=1101.024,315.439,417.740,179.154,17.355,151.880
C00766=1101.029,315.686,417.708,179.158,17.357,151.880
C00767=1101.038,316.071,417.659,179.163,17.361,151.880
C00768=1101.046,316.456,417.610,179.168,17.364,151.880
C00769=1101.055,316.841,417.561,179.173,17.367,151.879
C00770=1101.063,317.225,417.512,179.178,17.371,151.879
C00771=1101.069,317.473,417.481,179.181,17.374,151.879
C00772=1101.075,317.721,417.449,179.185,17.376,151.879
C00773=1101.080,317.969,417.417,179.188,17.378,151.879
C00774=1101.086,318.217,417.385,179.191,17.380,151.879
C00775=1101.092,318.464,417.353,179.195,17.383,151.879
C00776=1101.098,318.713,417.321,179.198,17.385,151.879
C00777=1101.103,318.961,417.290,179.201,17.387,151.878
C00778=1101.107,319.209,417.258,179.205,17.389,151.878
C00779=1101.113,319.457,417.226,179.208,17.392,151.878
C00780=1101.119,319.704,417.194,179.211,17.394,151.878
C00781=1101.125,319.952,417.162,179.214,17.396,151.878
C00782=1101.130,320.200,417.131,179.217,17.399,151.878
C00783=1101.136,320.448,417.099,179.221,17.401,151.878
C00784=1101.141,320.696,417.067,179.224,17.403,151.878
C00785=1101.147,320.944,417.035,179.227,17.405,151.878
C00786=1101.153,321.192,417.003,179.231,17.408,151.878
C00787=1101.159,321.440,416.971,179.234,17.410,151.878
C00788=1101.164,321.688,416.939,179.237,17.412,151.877
C00789=1101.170,321.935,416.906,179.240,17.415,151.877
C00790=1101.176,322.183,416.874,179.243,17.417,151.877
C00791=1101.181,322.431,416.842,179.248,17.420,151.877
C00792=1101.187,322.679,416.810,179.251,17.422,151.877
C00793=1101.193,322.927,416.779,179.254,17.425,151.877
C00794=1101.198,323.175,416.747,179.257,17.427,151.877
C00795=1101.204,323.423,416.714,179.261,17.429,151.877
C00796=1101.209,323.670,416.682,179.264,17.432,151.877
C00797=1101.215,323.918,416.650,179.267,17.434,151.877
C00798=1101.221,324.166,416.618,179.270,17.436,151.877
C00799=1101.227,324.414,416.586,179.273,17.439,151.876
C00800=1101.232,324.663,416.553,179.277,17.441,151.876
C00801=1101.238,324.909,416.521,179.280,17.443,151.876
C00802=1101.244,325.158,416.489,179.283,17.445,151.876
C00803=1101.250,325.406,416.457,179.286,17.448,151.876
C00804=1101.255,325.653,416.425,179.289,17.450,151.876
C00805=1101.261,325.901,416.392,179.294,17.453,151.876
C00806=1101.267,326.150,416.360,179.297,17.455,151.876
C00807=1101.272,326.396,416.328,179.300,17.458,151.876
C00808=1101.278,326.645,416.296,179.303,17.460,151.876
C00809=1101.284,326.893,416.263,179.306,17.463,151.876
C00810=1101.289,327.140,416.231,179.310,17.465,151.876
C00811=1101.295,327.388,416.199,179.313,17.467,151.876
C00812=1101.301,327.636,416.165,179.316,17.470,151.876
C00813=1101.307,327.884,416.133,179.319,17.472,151.876
C00814=1101.312,328.132,416.102,179.323,17.475,151.876
C00815=1101.318,328.380,416.069,179.326,17.478,151.875
C00816=1101.324,328.628,416.036,179.329,17.480,151.875
C00817=1101.330,328.876,416.003,179.333,17.482,151.875
C00818=1101.335,329.123,415.972,179.336,17.485,151.875
C00819=1101.344,329.501,415.921,179.341,17.488,151.875
C00820=1101.353,329.879,415.872,179.346,17.493,151.875
C00821=1101.362,330.256,415.822,179.351,17.496,151.875
C00822=1101.371,330.634,415.773,179.356,17.500,151.875
C00823=1101.376,330.882,415.740,179.359,17.503,151.875
C00824=1101.382,331.129,415.707,179.363,17.506,151.875
C00825=1101.388,331.377,415.675,179.366,17.508,151.875
C00826=1101.394,331.625,415.642,179.369,17.511,151.875
C00827=1101.400,331.872,415.609,179.372,17.513,151.875
C00828=1101.405,332.121,415.577,179.375,17.516,151.875
C00829=1101.411,332.368,415.544,179.378,17.518,151.875
C00830=1101.417,332.616,415.511,179.382,17.521,151.875
C00831=1101.423,332.864,415.478,179.385,17.524,151.875
C00832=1101.428,333.112,415.446,179.388,17.526,151.875
C00833=1101.433,333.360,415.412,179.391,17.529,151.875
C00834=1101.440,333.607,415.380,179.395,17.531,151.875
C00835=1101.445,333.855,415.346,179.397,17.534,151.875
C00836=1101.451,334.103,415.314,179.401,17.537,151.875
C00837=1101.457,334.351,415.281,179.405,17.540,151.875
C00838=1101.462,334.598,415.248,179.408,17.542,151.875
C00839=1101.468,334.846,415.215,179.411,17.545,151.875
C00840=1101.473,335.094,415.182,179.414,17.547,151.875
C00841=1101.479,335.342,415.149,179.418,17.551,151.875
C00842=1101.485,335.590,415.117,179.420,17.553,151.875
C00843=1101.491,335.838,415.083,179.424,17.556,151.875
C00844=1101.495,336.085,415.050,179.426,17.559,151.875
C00845=1101.502,336.333,415.017,179.430,17.562,151.875
C00846=1101.507,336.581,414.984,179.434,17.564,151.875
C00847=1101.513,336.828,414.951,179.436,17.567,151.875
C00848=1101.519,337.076,414.918,179.440,17.570,151.875
C00849=1101.525,337.324,414.885,179.443,17.573,151.875
C00850=1101.530,337.572,414.851,179.446,17.576,151.875
C00851=1101.537,337.819,414.819,179.449,17.578,151.875
C00852=1101.542,338.067,414.785,179.452,17.581,151.875
C00853=1101.548,338.315,414.752,179.455,17.584,151.876
C00854=1101.553,338.563,414.719,179.459,17.587,151.876
C00855=1101.560,338.811,414.686,179.462,17.590,151.876
C00856=1101.564,339.058,414.653,179.465,17.592,151.876
C00857=1101.570,339.305,414.619,179.469,17.596,151.876
C00858=1101.576,339.553,414.586,179.472,17.598,151.876
C00859=1101.581,339.801,414.552,179.475,17.601,151.876
C00860=1101.587,340.049,414.519,179.478,17.604,151.876
C00861=1101.593,340.297,414.485,179.482,17.607,151.876
C00862=1101.599,340.544,414.453,179.485,17.610,151.876
C00863=1101.605,340.792,414.419,179.487,17.613,151.876
C00864=1101.610,341.040,414.385,179.491,17.616,151.876
C00865=1101.616,341.288,414.352,179.494,17.619,151.876
C00866=1101.621,341.535,414.319,179.497,17.622,151.876
C00867=1101.627,341.783,414.285,179.500,17.624,151.877
C00868=1101.633,342.031,414.251,179.504,17.628,151.877
C00869=1101.638,342.279,414.218,179.507,17.630,151.877
C00870=1101.644,342.526,414.185,179.510,17.633,151.877
C00871=1101.653,342.898,414.134,179.515,17.638,151.877
C00872=1101.661,343.270,414.084,179.519,17.643,151.877
C00873=1101.670,343.641,414.033,179.524,17.647,151.877
C00874=1101.679,344.012,413.983,179.529,17.651,151.877
C00875=1101.684,344.260,413.950,179.532,17.655,151.878
C00876=1101.690,344.508,413.916,179.535,17.658,151.878
C00877=1101.696,344.755,413.882,179.538,17.661,151.878
C00878=1101.701,345.003,413.849,179.542,17.664,151.878
C00879=1101.707,345.250,413.815,179.545,17.667,151.878
C00880=1101.712,345.498,413.781,179.548,17.670,151.878
C00881=1101.718,345.746,413.747,179.551,17.673,151.878
C00882=1101.724,345.993,413.714,179.554,17.676,151.879
C00883=1101.729,346.241,413.680,179.557,17.679,151.879
C00884=1101.735,346.489,413.646,179.561,17.683,151.879
C00885=1101.741,346.737,413.612,179.564,17.685,151.879
C00886=1101.747,346.984,413.578,179.566,17.688,151.879
C00887=1101.753,347.232,413.544,179.570,17.692,151.879
C00888=1101.758,347.479,413.510,179.573,17.695,151.879
C00889=1101.763,347.727,413.476,179.576,17.699,151.880
C00890=1101.769,347.975,413.442,179.579,17.701,151.880
C00891=1101.775,348.222,413.408,179.582,17.704,151.880
C00892=1101.781,348.470,413.375,179.585,17.708,151.880
C00893=1101.786,348.717,413.340,179.588,17.711,151.880
C00894=1101.792,348.965,413.306,179.591,17.714,151.880
C00895=1101.798,349.213,413.272,179.595,17.717,151.881
C00896=1101.804,349.461,413.239,179.597,17.721,151.881
C00897=1101.810,349.708,413.204,179.601,17.724,151.881
C00898=1101.815,349.955,413.170,179.604,17.727,151.881
C00899=1101.821,350.203,413.136,179.607,17.731,151.881
C00900=1101.826,350.451,413.102,179.610,17.734,151.882
C00901=1101.831,350.698,413.068,179.613,17.737,151.882
C00902=1101.838,350.946,413.033,179.617,17.741,151.882
C00903=1101.844,351.193,412.999,179.619,17.743,151.882
C00904=1101.849,351.441,412.965,179.623,17.747,151.882
C00905=1101.855,351.688,412.931,179.626,17.750,151.883
C00906=1101.860,351.936,412.897,179.629,17.754,151.883
C00907=1101.867,352.184,412.863,179.632,17.757,151.883
C00908=1101.872,352.432,412.828,179.635,17.760,151.883
C00909=1101.878,352.679,412.794,179.638,17.764,151.883
C00910=1101.883,352.926,412.760,179.641,17.767,151.884
C00911=1101.889,353.174,412.725,179.644,17.771,151.884
C00912=1101.895,353.422,412.691,179.647,17.774,151.884
C00913=1101.901,353.669,412.657,179.650,17.778,151.884
C00914=1101.906,353.917,412.622,179.653,17.781,151.884
C00915=1101.912,354.164,412.588,179.657,17.784,151.885
C00916=1101.917,354.412,412.554,179.659,17.788,151.885
C00917=1101.923,354.660,412.519,179.663,17.791,151.885
C00918=1101.929,354.907,412.485,179.666,17.795,151.885
C00919=1101.934,355.155,412.451,179.669,17.798,151.886
C00920=1101.940,355.402,412.415,179.672,17.802,151.886
C00921=1101.946,355.650,412.381,179.675,17.805,151.886
C00922=1101.951,355.897,412.346,179.678,17.808,151.886
C00923=1101.960,356.271,412.295,179.683,17.814,151.887
C00924=1101.969,356.644,412.242,179.687,17.820,151.887
C00925=1101.977,357.019,412.190,179.691,17.824,151.888
C00926=1101.986,357.392,412.137,179.696,17.830,151.888
C00927=1101.991,357.639,412.103,179.699,17.834,151.889
C00928=1101.997,357.888,412.068,179.702,17.837,151.889
C00929=1102.003,358.134,412.033,179.705,17.841,151.889
C00930=1102.008,358.382,411.999,179.708,17.844,151.889
C00931=1102.015,358.630,411.964,179.711,17.848,151.890
C00932=1102.020,358.877,411.929,179.714,17.852,151.890
C00933=1102.025,359.124,411.894,179.717,17.855,151.890
C00934=1102.032,359.372,411.860,179.720,17.859,151.891
C00935=1102.037,359.619,411.824,179.723,17.863,151.891
C00936=1102.043,359.867,411.790,179.726,17.866,151.891
C00937=1102.049,360.115,411.755,179.729,17.870,151.891
C00938=1102.054,360.362,411.720,179.733,17.874,151.892
C00939=1102.061,360.610,411.686,179.735,17.877,151.892
C00940=1102.066,360.857,411.650,179.738,17.881,151.892
C00941=1102.071,361.104,411.616,179.741,17.885,151.893
C00942=1102.077,361.352,411.580,179.744,17.888,151.893
C00943=1102.083,361.599,411.546,179.747,17.892,151.893
C00944=1102.089,361.846,411.510,179.750,17.896,151.894
C00945=1102.094,362.095,411.475,179.754,17.900,151.894
C00946=1102.100,362.342,411.440,179.756,17.904,151.895
C00947=1102.106,362.589,411.406,179.759,17.907,151.895
C00948=1102.112,362.837,411.370,179.762,17.911,151.895
C00949=1102.117,363.084,411.335,179.765,17.915,151.896
C00950=1102.123,363.332,411.300,179.768,17.919,151.896
C00951=1102.129,363.578,411.265,179.771,17.923,151.896
C00952=1102.135,363.826,411.229,179.774,17.927,151.897
C00953=1102.140,364.074,411.195,179.777,17.930,151.897
C00954=1102.146,364.321,411.159,179.780,17.934,151.897
C00955=1102.152,364.568,411.124,179.783,17.938,151.898
C00956=1102.158,364.816,411.090,179.785,17.942,151.898
C00957=1102.164,365.063,411.054,179.789,17.946,151.898
C00958=1102.169,365.310,411.019,179.791,17.950,151.899
C00959=1102.175,365.559,410.984,179.794,17.954,151.899
C00960=1102.180,365.806,410.948,179.798,17.958,151.900
C00961=1102.186,366.053,410.912,179.800,17.962,151.900
C00962=1102.192,366.300,410.877,179.803,17.966,151.901
C00963=1102.197,366.547,410.842,179.806,17.970,151.901
C00964=1102.203,366.795,410.806,179.809,17.974,151.901
C00965=1102.208,367.042,410.771,179.812,17.978,151.902
C00966=1102.214,367.290,410.736,179.815,17.982,151.902
C00967=1102.220,367.537,410.700,179.818,17.986,151.903
C00968=1102.226,367.785,410.664,179.821,17.990,151.903
C00969=1102.231,368.032,410.629,179.824,17.994,151.904
C00970=1102.237,368.279,410.593,179.826,17.998,151.904
C00971=1102.243,368.526,410.558,179.829,18.002,151.904
C00972=1102.249,368.774,410.522,179.833,18.007,151.905
C00973=1102.254,369.021,410.487,179.835,18.010,151.905
C00974=1102.260,369.269,410.451,179.838,18.014,151.906
C00975=1102.269,369.657,410.396,179.842,18.021,151.907
C00976=1102.278,370.046,410.339,179.847,18.028,151.907
C00977=1102.287,370.434,410.283,179.851,18.034,151.908
C00978=1102.296,370.823,410.227,179.856,18.041,151.909
C00979=1102.301,371.070,410.192,179.859,18.045,151.909
C00980=1102.307,371.318,410.156,179.862,18.049,151.910
C00981=1102.313,371.565,410.120,179.865,18.054,151.910
C00982=1102.319,371.813,410.085,179.868,18.058,151.911
C00983=1102.325,372.060,410.049,179.870,18.062,151.911
C00984=1102.330,372.307,410.013,179.873,18.066,151.912
C00985=1102.336,372.554,409.977,179.876,18.071,151.912
C00986=1102.341,372.802,409.941,179.879,18.075,151.913
C00987=1102.347,373.049,409.905,179.881,18.079,151.913
C00988=1102.353,373.297,409.870,179.884,18.084,151.914
C00989=1102.359,373.543,409.834,179.887,18.088,151.914
C00990=1102.365,373.791,409.798,179.891,18.092,151.915
C00991=1102.371,374.039,409.762,179.893,18.096,151.915
C00992=1102.376,374.285,409.726,179.896,18.101,151.916
C00993=1102.382,374.533,409.690,179.899,18.105,151.916
C00994=1102.387,374.780,409.654,179.902,18.110,151.917
C00995=1102.393,375.027,409.617,179.904,18.114,151.918
C00996=1102.399,375.275,409.582,179.907,18.118,151.918
C00997=1102.405,375.521,409.546,179.910,18.123,151.919
C00998=1102.410,375.769,409.509,179.913,18.128,151.919
C00999=1102.416,376.017,409.474,179.915,18.133,151.920
C01000=1102.422,376.263,409.437,179.918,18.137,151.920
C01001=1102.427,376.511,409.401,179.920,18.141,151.921
C01002=1102.433,376.758,409.365,179.924,18.146,151.922
C01003=1102.438,377.006,409.329,179.926,18.150,151.922
C01004=1102.444,377.253,409.292,179.929,18.155,151.923
C01005=1102.450,377.500,409.257,179.932,18.160,151.923
C01006=1102.455,377.747,409.220,179.934,18.164,151.924
C01007=1102.462,377.994,409.183,179.937,18.168,151.925
C01008=1102.467,378.241,409.147,179.940,18.173,151.925
C01009=1102.473,378.488,409.111,179.943,18.178,151.926
C01010=1102.479,378.736,409.075,179.946,18.183,151.926
C01011=1102.484,378.983,409.039,179.949,18.188,151.927
C01012=1102.490,379.230,409.002,179.951,18.192,151.928
C01013=1102.495,379.478,408.966,179.954,18.196,151.928
C01014=1102.502,379.725,408.929,179.956,18.201,151.929
C01015=1102.507,379.971,408.893,179.959,18.206,151.930
C01016=1102.513,380.219,408.857,179.962,18.211,151.930
C01017=1102.518,380.467,408.820,179.965,18.216,151.931
C01018=1102.525,380.714,408.784,179.967,18.221,151.932
C01019=1102.530,380.960,408.747,179.970,18.225,151.932
C01020=1102.536,381.208,408.711,179.973,18.230,151.933
C01021=1102.541,381.455,408.674,179.975,18.234,151.934
C01022=1102.548,381.702,408.638,179.978,18.239,151.934
C01023=1102.553,381.950,408.601,179.981,18.244,151.935
C01024=1102.559,382.196,408.565,179.983,18.249,151.935
C01025=1102.565,382.443,408.527,179.986,18.254,151.936
C01026=1102.571,382.690,408.491,179.989,18.259,151.937
C01027=1102.580,383.106,408.430,179.993,18.267,151.938
C01028=1102.590,383.522,408.368,179.998,18.276,151.939
C01029=1102.599,383.937,408.306,-179.998,18.284,151.940
C01030=1102.608,384.353,408.244,-179.993,18.292,151.942
C01031=1102.614,384.600,408.207,-179.991,18.297,151.942
C01032=1102.620,384.847,408.171,-179.988,18.302,151.943
C01033=1102.626,385.095,408.134,-179.985,18.307,151.944
C01034=1102.632,385.342,408.097,-179.983,18.312,151.945
C01035=1102.637,385.589,408.060,-179.980,18.317,151.945
C01036=1102.643,385.836,408.024,-179.977,18.322,151.946
C01037=1102.648,386.083,407.987,-179.975,18.327,151.947
C01038=1102.654,386.330,407.949,-179.972,18.333,151.948
C01039=1102.660,386.577,407.912,-179.970,18.338,151.948
C01040=1102.666,386.824,407.875,-179.967,18.343,151.949
C01041=1102.671,387.071,407.839,-179.965,18.348,151.950
C01042=1102.677,387.318,407.802,-179.962,18.353,151.951
C01043=1102.683,387.565,407.765,-179.959,18.358,151.952
C01044=1102.688,387.812,407.727,-179.957,18.363,151.952
C01045=1102.694,388.060,407.690,-179.953,18.370,151.953
C01046=1102.700,388.307,407.653,-179.951,18.375,151.954
C01047=1102.706,388.553,407.616,-179.948,18.380,151.955
C01048=1102.712,388.801,407.578,-179.946,18.385,151.956
C01049=1102.717,389.048,407.541,-179.943,18.390,151.956
C01050=1102.723,389.295,407.504,-179.941,18.396,151.957
C01051=1102.728,389.542,407.467,-179.938,18.401,151.958
C01052=1102.734,389.789,407.430,-179.936,18.406,151.959
C01053=1102.741,390.035,407.393,-179.933,18.411,151.960
C01054=1102.746,390.283,407.356,-179.931,18.417,151.961
C01055=1102.752,390.530,407.319,-179.928,18.422,151.961
C01056=1102.758,390.777,407.281,-179.926,18.427,151.962
C01057=1102.763,391.024,407.244,-179.923,18.433,151.963
C01058=1102.769,391.271,407.206,-179.921,18.438,151.964
C01059=1102.775,391.518,407.169,-179.917,18.444,151.965
C01060=1102.781,391.765,407.131,-179.915,18.450,151.966
C01061=1102.786,392.012,407.094,-179.913,18.455,151.967
C01062=1102.792,392.259,407.057,-179.910,18.460,151.968
C01063=1102.798,392.507,407.019,-179.908,18.466,151.969
C01064=1102.804,392.753,406.982,-179.905,18.471,151.969
C01065=1102.810,393.001,406.944,-179.903,18.477,151.970
C01066=1102.816,393.248,406.907,-179.901,18.482,151.971
C01067=1102.821,393.495,406.870,-179.897,18.488,151.972
C01068=1102.827,393.742,406.832,-179.895,18.494,151.973
C01069=1102.833,393.989,406.794,-179.893,18.499,151.974
C01070=1102.839,394.236,406.757,-179.890,18.505,151.975
C01071=1102.844,394.483,406.719,-179.888,18.511,151.976
C01072=1102.850,394.730,406.681,-179.886,18.516,151.977
C01073=1102.855,394.977,406.644,-179.883,18.522,151.978
C01074=1102.861,395.224,406.606,-179.880,18.528,151.979
C01075=1102.867,395.471,406.568,-179.878,18.534,151.980
C01076=1102.873,395.718,406.531,-179.876,18.540,151.981
C01077=1102.878,395.965,406.493,-179.873,18.545,151.982
C01078=1102.884,396.212,406.455,-179.871,18.551,151.983
C01079=1102.890,396.426,406.422,-179.869,18.556,151.984
C01080=1102.894,396.641,406.390,-179.867,18.561,151.984
C01081=1102.899,396.854,406.357,-179.864,18.566,151.985
C01082=1102.904,397.068,406.324,-179.862,18.572,151.986
C01083=1102.909,397.282,406.291,-179.860,18.577,151.987
C01084=1102.914,397.496,406.259,-179.858,18.582,151.988
C01085=1102.919,397.710,406.226,-179.856,18.587,151.989
C01086=1102.924,397.923,406.193,-179.854,18.592,151.990
C01087=1102.930,398.171,406.155,-179.851,18.598,151.991
C01088=1102.935,398.418,406.117,-179.849,18.604,151.992
C01089=1102.941,398.665,406.079,-179.847,18.610,151.993
C01090=1102.947,398.911,406.041,-179.844,18.616,151.994
C01091=1102.952,399.159,406.003,-179.842,18.622,151.995
C01092=1102.959,399.407,405.965,-179.840,18.628,151.996
C01093=1102.964,399.653,405.927,-179.837,18.634,151.997
C01094=1102.970,399.900,405.889,-179.835,18.640,151.998
C01095=1102.975,400.147,405.851,-179.833,18.646,151.999
C01096=1102.981,400.394,405.813,-179.831,18.652,152.000
C01097=1102.987,400.641,405.774,-179.828,18.659,152.001
C01098=1102.993,400.888,405.736,-179.826,18.665,152.003
C01099=1102.999,401.135,405.698,-179.824,18.671,152.004
C01100=1103.004,401.381,405.660,-179.821,18.678,152.005
C01101=1103.010,401.629,405.622,-179.819,18.684,152.006
C01102=1103.016,401.876,405.584,-179.817,18.690,152.007
C01103=1103.021,402.123,405.546,-179.814,18.696,152.008
C01104=1103.027,402.370,405.508,-179.812,18.703,152.009
C01105=1103.033,402.617,405.468,-179.809,18.709,152.010
C01106=1103.039,402.864,405.431,-179.807,18.715,152.012
C01107=1103.044,403.111,405.392,-179.805,18.721,152.013
C01108=1103.050,403.358,405.354,-179.802,18.728,152.014
C01109=1103.056,403.605,405.316,-179.800,18.734,152.015
C01110=1103.061,403.852,405.277,-179.797,18.741,152.016
C01111=1103.067,404.098,405.239,-179.795,18.747,152.017
C01112=1103.073,404.346,405.200,-179.794,18.754,152.019
C01113=1103.079,404.592,405.162,-179.791,18.760,152.020
C01114=1103.085,404.839,405.123,-179.789,18.767,152.021
C01115=1103.090,405.087,405.085,-179.786,18.774,152.022
C01116=1103.097,405.333,405.046,-179.784,18.780,152.023
C01117=1103.102,405.580,405.008,-179.781,18.787,152.025
C01118=1103.108,405.827,404.968,-179.780,18.793,152.026
C01119=1103.114,406.074,404.931,-179.777,18.800,152.027
C01120=1103.119,406.322,404.892,-179.775,18.806,152.028
C01121=1103.125,406.568,404.853,-179.773,18.814,152.030
C01122=1103.131,406.815,404.815,-179.771,18.820,152.031
C01123=1103.137,407.062,404.776,-179.768,18.827,152.032
C01124=1103.142,407.309,404.737,-179.766,18.833,152.033
C01125=1103.148,407.556,404.698,-179.764,18.841,152.035
C01126=1103.153,407.803,404.660,-179.762,18.847,152.036
C01127=1103.159,408.050,404.621,-179.759,18.854,152.037
C01128=1103.166,408.297,404.582,-179.758,18.861,152.039
C01129=1103.171,408.544,404.543,-179.755,18.868,152.040
C01130=1103.176,408.790,404.504,-179.752,18.875,152.041
C01131=1103.182,409.038,404.466,-179.751,18.882,152.043
C01132=1103.187,409.284,404.426,-179.748,18.889,152.044
C01133=1103.194,409.532,404.387,-179.746,18.895,152.045
C01134=1103.199,409.778,404.349,-179.744,18.903,152.047
C01135=1103.205,409.992,404.315,-179.742,18.909,152.048
C01136=1103.209,410.206,404.282,-179.740,18.915,152.049
C01137=1103.215,410.420,404.247,-179.738,18.921,152.050
C01138=1103.219,410.634,404.214,-179.737,18.927,152.051
C01139=1103.224,410.847,404.180,-179.735,18.933,152.053
C01140=1103.229,411.062,404.146,-179.733,18.939,152.054
C01141=1103.234,411.275,404.112,-179.731,18.946,152.055
C01142=1103.239,411.490,404.079,-179.729,18.952,152.056
C01143=1103.245,411.736,404.040,-179.727,18.960,152.058
C01144=1103.251,411.983,404.000,-179.725,18.966,152.059
C01145=1103.256,412.230,403.961,-179.723,18.974,152.061
C01146=1103.262,412.477,403.922,-179.720,18.981,152.062
C01147=1103.268,412.723,403.883,-179.718,18.989,152.063
C01148=1103.274,412.970,403.843,-179.716,18.996,152.065
C01149=1103.279,413.217,403.804,-179.714,19.003,152.066
C01150=1103.285,413.464,403.765,-179.712,19.011,152.068
C01151=1103.291,413.710,403.726,-179.710,19.018,152.069
C01152=1103.297,413.957,403.686,-179.708,19.025,152.071
C01153=1103.302,414.204,403.647,-179.706,19.033,152.072
C01154=1103.308,414.451,403.608,-179.703,19.041,152.074
C01155=1103.314,414.698,403.568,-179.701,19.048,152.075
C01156=1103.320,414.945,403.529,-179.699,19.055,152.077
C01157=1103.326,415.192,403.490,-179.697,19.063,152.078
C01158=1103.331,415.438,403.451,-179.695,19.070,152.080
C01159=1103.338,415.685,403.411,-179.693,19.078,152.081
C01160=1103.343,415.933,403.371,-179.690,19.086,152.083
C01161=1103.348,416.179,403.332,-179.689,19.093,152.084
C01162=1103.355,416.426,403.292,-179.687,19.101,152.086
C01163=1103.361,416.673,403.253,-179.684,19.108,152.087
C01164=1103.366,416.919,403.214,-179.682,19.116,152.089
C01165=1103.372,417.166,403.174,-179.680,19.124,152.090
C01166=1103.377,417.412,403.134,-179.678,19.132,152.092
C01167=1103.383,417.660,403.094,-179.676,19.140,152.094
C01168=1103.389,417.906,403.055,-179.675,19.148,152.095
C01169=1103.395,418.153,403.016,-179.673,19.156,152.097
C01170=1103.401,418.400,402.975,-179.670,19.164,152.099
C01171=1103.406,418.646,402.936,-179.668,19.172,152.100
C01172=1103.412,418.893,402.896,-179.666,19.180,152.102
C01173=1103.418,419.140,402.856,-179.664,19.188,152.103
C01174=1103.423,419.387,402.817,-179.662,19.196,152.105
C01175=1103.430,419.633,402.777,-179.660,19.204,152.107
C01176=1103.434,419.880,402.737,-179.658,19.212,152.108
C01177=1103.441,420.127,402.697,-179.656,19.220,152.110
C01178=1103.447,420.374,402.657,-179.654,19.228,152.112
C01179=1103.453,420.621,402.617,-179.652,19.236,152.113
C01180=1103.458,420.867,402.578,-179.650,19.244,152.115
C01181=1103.464,421.114,402.537,-179.648,19.252,152.117
C01182=1103.470,421.361,402.497,-179.646,19.261,152.119
C01183=1103.475,421.607,402.458,-179.644,19.269,152.120
C01184=1103.482,421.853,402.417,-179.642,19.277,152.122
C01185=1103.487,422.101,402.377,-179.640,19.286,152.124
C01186=1103.494,422.347,402.337,-179.639,19.294,152.126
C01187=1103.498,422.594,402.298,-179.637,19.302,152.127
C01188=1103.505,422.841,402.257,-179.635,19.311,152.129
C01189=1103.510,423.087,402.217,-179.633,19.319,152.131
C01190=1103.517,423.334,402.177,-179.631,19.328,152.133
C01191=1103.522,423.555,402.141,-179.629,19.336,152.134
C01192=1103.526,423.775,402.105,-179.628,19.343,152.136
C01193=1103.531,423.996,402.069,-179.626,19.351,152.138
C01194=1103.536,424.216,402.033,-179.624,19.358,152.139
C01195=1103.542,424.437,401.997,-179.622,19.366,152.141
C01196=1103.547,424.657,401.961,-179.621,19.374,152.143
C01197=1103.552,424.878,401.925,-179.619,19.382,152.144
C01198=1103.558,425.099,401.889,-179.618,19.390,152.146
C01199=1103.563,425.345,401.849,-179.616,19.398,152.148
C01200=1103.569,425.591,401.808,-179.614,19.407,152.150
C01201=1103.575,425.838,401.768,-179.612,19.416,152.152
C01202=1103.580,426.085,401.727,-179.610,19.425,152.153
C01203=1103.587,426.331,401.687,-179.608,19.434,152.155
C01204=1103.592,426.577,401.646,-179.607,19.443,152.157
C01205=1103.597,426.824,401.606,-179.605,19.451,152.159
C01206=1103.604,427.071,401.566,-179.602,19.461,152.161
C01207=1103.609,427.318,401.525,-179.601,19.469,152.163
C01208=1103.615,427.564,401.484,-179.599,19.479,152.165
C01209=1103.621,427.810,401.444,-179.598,19.487,152.167
C01210=1103.626,428.057,401.404,-179.595,19.497,152.169
C01211=1103.632,428.304,401.363,-179.594,19.506,152.171
C01212=1103.639,428.550,401.323,-179.592,19.515,152.173
C01213=1103.644,428.797,401.282,-179.591,19.524,152.175
C01214=1103.650,429.044,401.241,-179.588,19.534,152.177
C01215=1103.656,429.290,401.200,-179.587,19.542,152.179
C01216=1103.662,429.537,401.160,-179.585,19.552,152.181
C01217=1103.667,429.783,401.119,-179.583,19.561,152.183
C01218=1103.673,430.030,401.078,-179.582,19.571,152.185
C01219=1103.679,430.276,401.037,-179.580,19.580,152.187
C01220=1103.684,430.523,400.996,-179.578,19.590,152.189
C01221=1103.690,430.770,400.956,-179.577,19.599,152.191
C01222=1103.696,431.016,400.914,-179.575,19.608,152.194
C01223=1103.702,431.262,400.874,-179.573,19.618,152.196
C01224=1103.708,431.509,400.833,-179.572,19.628,152.198
C01225=1103.714,431.755,400.792,-179.570,19.637,152.200
C01226=1103.720,432.002,400.751,-179.568,19.647,152.202
C01227=1103.725,432.248,400.710,-179.567,19.656,152.204
C01228=1103.731,432.494,400.669,-179.566,19.666,152.206
C01229=1103.737,432.741,400.628,-179.564,19.676,152.209
C01230=1103.742,432.988,400.587,-179.562,19.686,152.211
C01231=1103.748,433.234,400.545,-179.560,19.696,152.213
C01232=1103.754,433.481,400.505,-179.559,19.705,152.215
C01233=1103.760,433.727,400.463,-179.557,19.716,152.217
C01234=1103.765,433.974,400.423,-179.556,19.725,152.220
C01235=1103.771,434.220,400.381,-179.554,19.736,152.222
C01236=1103.777,434.467,400.340,-179.552,19.745,152.224
C01237=1103.783,434.713,400.299,-179.551,19.756,152.227
C01238=1103.789,434.959,400.257,-179.550,19.766,152.229
C01239=1103.794,435.206,400.217,-179.547,19.776,152.231
C01240=1103.800,435.452,400.175,-179.546,19.786,152.233
C01241=1103.806,435.699,400.133,-179.545,19.796,152.236
C01242=1103.812,435.945,400.092,-179.544,19.806,152.238
C01243=1103.817,436.192,400.051,-179.542,19.817,152.240
C01244=1103.823,436.438,400.009,-179.541,19.827,152.243
C01245=1103.829,436.684,399.968,-179.539,19.837,152.245
C01246=1103.835,436.930,399.927,-179.538,19.848,152.248
C01247=1103.844,437.337,399.858,-179.535,19.865,152.252
C01248=1103.854,437.744,399.789,-179.533,19.882,152.256
C01249=1103.864,438.151,399.720,-179.530,19.900,152.260
C01250=1103.873,438.558,399.653,-179.528,19.917,152.264
C01251=1103.878,438.805,399.611,-179.527,19.928,152.266
C01252=1103.885,439.052,399.569,-179.526,19.939,152.269
C01253=1103.891,439.298,399.527,-179.524,19.950,152.271
C01254=1103.897,439.544,399.486,-179.523,19.960,152.274
C01255=1103.902,439.791,399.444,-179.521,19.971,152.276
C01256=1103.908,440.036,399.402,-179.520,19.982,152.279
C01257=1103.914,440.282,399.360,-179.519,19.992,152.281
C01258=1103.920,440.529,399.319,-179.517,20.004,152.284
C01259=1103.925,440.775,399.277,-179.516,20.015,152.286
C01260=1103.932,441.022,399.235,-179.515,20.025,152.289
C01261=1103.938,441.268,399.193,-179.514,20.037,152.291
C01262=1103.943,441.515,399.151,-179.512,20.048,152.294
C01263=1103.949,441.760,399.109,-179.511,20.059,152.297
C01264=1103.954,442.007,399.067,-179.510,20.070,152.299
C01265=1103.960,442.253,399.026,-179.509,20.082,152.302
C01266=1103.966,442.499,398.983,-179.507,20.093,152.305
C01267=1103.972,442.746,398.941,-179.506,20.105,152.307
C01268=1103.978,442.992,398.899,-179.505,20.115,152.310
C01269=1103.984,443.238,398.857,-179.504,20.127,152.313
C01270=1103.989,443.484,398.815,-179.503,20.139,152.316
C01271=1103.995,443.731,398.773,-179.501,20.150,152.318
C01272=1104.001,443.977,398.731,-179.501,20.162,152.321
C01273=1104.007,444.223,398.689,-179.499,20.173,152.324
C01274=1104.013,444.469,398.646,-179.499,20.185,152.327
C01275=1104.019,444.716,398.604,-179.499,20.196,152.330
C01276=1104.024,444.961,398.562,-179.498,20.207,152.332
C01277=1104.030,445.209,398.519,-179.498,20.219,152.335
C01278=1104.036,445.454,398.477,-179.499,20.230,152.338
C01279=1104.041,445.701,398.435,-179.498,20.241,152.341
C01280=1104.048,445.946,398.393,-179.499,20.252,152.344
C01281=1104.053,446.194,398.350,-179.499,20.264,152.347
C01282=1104.059,446.439,398.308,-179.499,20.275,152.350
C01283=1104.065,446.686,398.266,-179.500,20.286,152.353
C01284=1104.071,446.932,398.223,-179.501,20.298,152.356
C01285=1104.077,447.178,398.180,-179.501,20.309,152.359
C01286=1104.082,447.425,398.138,-179.502,20.320,152.362
C01287=1104.088,447.670,398.096,-179.503,20.332,152.365
C01288=1104.094,447.917,398.053,-179.504,20.343,152.368
C01289=1104.099,448.163,398.011,-179.505,20.354,152.371
C01290=1104.105,448.409,397.968,-179.507,20.365,152.374
C01291=1104.112,448.656,397.926,-179.508,20.377,152.377
C01292=1104.117,448.902,397.884,-179.509,20.388,152.380
C01293=1104.122,449.148,397.841,-179.511,20.399,152.383
C01294=1104.129,449.395,397.798,-179.513,20.410,152.386
C01295=1104.135,449.641,397.756,-179.515,20.421,152.390
C01296=1104.140,449.887,397.713,-179.516,20.432,152.393
C01297=1104.146,450.133,397.670,-179.518,20.443,152.396
C01298=1104.152,450.379,397.628,-179.520,20.455,152.399
C01299=1103.749,450.372,397.497,-179.594,20.682,152.469
C01300=1103.743,450.126,397.540,-179.592,20.671,152.466
C01301=1103.737,449.879,397.581,-179.591,20.660,152.463
C01302=1103.731,449.633,397.625,-179.588,20.648,152.460
C01303=1103.726,449.387,397.667,-179.586,20.637,152.457
C01304=1103.720,449.141,397.710,-179.585,20.626,152.454
C01305=1103.714,448.895,397.753,-179.584,20.614,152.451
C01306=1103.708,448.648,397.795,-179.582,20.603,152.447
C01307=1103.702,448.402,397.838,-179.581,20.592,152.444
C01308=1103.696,448.156,397.881,-179.580,20.581,152.441
C01309=1103.691,447.910,397.923,-179.578,20.569,152.438
C01310=1103.685,447.663,397.966,-179.578,20.558,152.435
C01311=1103.679,447.417,398.008,-179.577,20.546,152.432
C01312=1103.673,447.171,398.051,-179.575,20.536,152.429
C01313=1103.667,446.924,398.093,-179.575,20.524,152.426
C01314=1103.662,446.678,398.136,-179.574,20.513,152.423
C01315=1103.656,446.433,398.178,-179.574,20.502,152.420
C01316=1103.650,446.185,398.221,-179.574,20.490,152.417
C01317=1103.644,445.939,398.263,-179.573,20.479,152.414
C01318=1103.638,445.694,398.305,-179.574,20.467,152.411
C01319=1103.633,445.447,398.348,-179.573,20.456,152.408
C01320=1103.627,445.201,398.391,-179.573,20.444,152.405
C01321=1103.621,444.955,398.432,-179.574,20.432,152.402
C01322=1103.615,444.709,398.475,-179.574,20.421,152.400
C01323=1103.609,444.462,398.517,-179.575,20.410,152.397
C01324=1103.603,444.216,398.559,-179.575,20.398,152.394
C01325=1103.598,443.969,398.602,-179.576,20.386,152.391
C01326=1103.592,443.724,398.644,-179.577,20.375,152.388
C01327=1103.587,443.477,398.686,-179.578,20.363,152.386
C01328=1103.580,443.231,398.728,-179.580,20.352,152.383
C01329=1103.575,442.984,398.770,-179.580,20.341,152.380
C01330=1103.568,442.739,398.813,-179.582,20.329,152.377
C01331=1103.563,442.492,398.855,-179.583,20.317,152.375
C01332=1103.557,442.246,398.896,-179.584,20.306,152.372
C01333=1103.551,442.000,398.939,-179.585,20.295,152.369
C01334=1103.545,441.753,398.981,-179.587,20.283,152.367
C01335=1103.540,441.507,399.023,-179.588,20.272,152.364
C01336=1103.534,441.261,399.065,-179.590,20.261,152.361
C01337=1103.528,441.015,399.106,-179.591,20.250,152.359
C01338=1103.522,440.769,399.148,-179.592,20.239,152.356
C01339=1103.516,440.522,399.190,-179.594,20.227,152.354
C01340=1103.510,440.276,399.233,-179.595,20.216,152.351
C01341=1103.504,440.030,399.274,-179.596,20.205,152.349
C01342=1103.498,439.783,399.316,-179.598,20.194,152.346
C01343=1103.493,439.537,399.357,-179.600,20.183,152.343
C01344=1103.487,439.291,399.399,-179.600,20.173,152.341
C01345=1103.481,439.044,399.441,-179.602,20.162,152.338
C01346=1103.475,438.798,399.483,-179.603,20.151,152.336
C01347=1103.469,438.551,399.524,-179.605,20.140,152.333
C01348=1103.459,438.150,399.592,-179.607,20.123,152.329
C01349=1103.450,437.748,399.660,-179.610,20.105,152.325
C01350=1103.441,437.347,399.728,-179.612,20.088,152.321
C01351=1103.432,436.945,399.796,-179.614,20.071,152.318
C01352=1103.426,436.699,399.837,-179.616,20.060,152.315
C01353=1103.420,436.453,399.879,-179.617,20.050,152.313
C01354=1103.414,436.207,399.920,-179.619,20.040,152.310
C01355=1103.408,435.961,399.961,-179.620,20.029,152.308
C01356=1103.402,435.714,400.003,-179.622,20.019,152.306
C01357=1103.397,435.467,400.044,-179.623,20.009,152.303
C01358=1103.391,435.221,400.086,-179.625,19.998,152.301
C01359=1103.385,434.975,400.127,-179.627,19.988,152.299
C01360=1103.379,434.729,400.169,-179.628,19.978,152.296
C01361=1103.373,434.482,400.209,-179.630,19.967,152.294
C01362=1103.367,434.236,400.251,-179.631,19.957,152.292
C01363=1103.361,433.989,400.292,-179.633,19.948,152.290
C01364=1103.356,433.743,400.333,-179.635,19.937,152.287
C01365=1103.351,433.496,400.375,-179.636,19.928,152.285
C01366=1103.344,433.250,400.416,-179.638,19.917,152.283
C01367=1103.338,433.003,400.457,-179.639,19.908,152.281
C01368=1103.332,432.757,400.498,-179.641,19.898,152.278
C01369=1103.327,432.510,400.539,-179.643,19.888,152.276
C01370=1103.321,432.264,400.580,-179.645,19.878,152.274
C01371=1103.315,432.017,400.621,-179.646,19.868,152.272
C01372=1103.309,431.771,400.663,-179.648,19.859,152.270
C01373=1103.304,431.524,400.703,-179.650,19.849,152.267
C01374=1103.298,431.278,400.745,-179.651,19.840,152.265
C01375=1103.293,431.032,400.785,-179.653,19.829,152.263
C01376=1103.287,430.785,400.826,-179.655,19.820,152.261
C01377=1103.281,430.539,400.867,-179.656,19.811,152.259
C01378=1103.275,430.292,400.908,-179.659,19.801,152.257
C01379=1103.269,430.046,400.948,-179.660,19.791,152.255
C01380=1103.263,429.799,400.990,-179.662,19.782,152.253
C01381=1103.257,429.552,401.030,-179.664,19.773,152.251
C01382=1103.252,429.306,401.071,-179.665,19.763,152.248
C01383=1103.246,429.059,401.113,-179.667,19.754,152.247
C01384=1103.239,428.813,401.153,-179.669,19.744,152.244
C01385=1103.234,428.567,401.193,-179.671,19.735,152.242
C01386=1103.229,428.320,401.234,-179.672,19.726,152.240
C01387=1103.223,428.073,401.275,-179.674,19.717,152.238
C01388=1103.216,427.827,401.315,-179.676,19.708,152.236
C01389=1103.211,427.580,401.356,-179.678,19.698,152.234
C01390=1103.205,427.334,401.397,-179.680,19.690,152.232
C01391=1103.199,427.087,401.437,-179.681,19.681,152.230
C01392=1103.193,426.840,401.478,-179.684,19.671,152.229
C01393=1103.188,426.594,401.518,-179.685,19.662,152.227
C01394=1103.182,426.348,401.558,-179.687,19.654,152.225
C01395=1103.176,426.101,401.599,-179.689,19.644,152.223
C01396=1103.170,425.854,401.640,-179.690,19.636,152.221
C01397=1103.164,425.607,401.680,-179.693,19.626,152.219
C01398=1103.159,425.361,401.720,-179.695,19.618,152.217
C01399=1103.153,425.115,401.761,-179.696,19.609,152.215
C01400=1103.147,424.894,401.797,-179.698,19.601,152.213
C01401=1103.142,424.673,401.833,-179.700,19.593,152.212
C01402=1103.138,424.451,401.869,-179.701,19.586,152.210
C01403=1103.132,424.231,401.905,-179.703,19.578,152.208
C01404=1103.127,424.010,401.942,-179.705,19.570,152.207
C01405=1103.122,423.790,401.977,-179.707,19.562,152.205
C01406=1103.116,423.569,402.014,-179.708,19.554,152.203
C01407=1103.112,423.348,402.050,-179.710,19.546,152.202
C01408=1103.106,423.101,402.089,-179.712,19.538,152.200
C01409=1103.100,422.854,402.130,-179.714,19.529,152.198
C01410=1103.094,422.608,402.170,-179.716,19.521,152.196
C01411=1103.089,422.361,402.210,-179.718,19.513,152.195
C01412=1103.083,422.114,402.250,-179.720,19.504,152.193
C01413=1103.076,421.868,402.290,-179.722,19.496,152.191
C01414=1103.072,421.621,402.330,-179.724,19.487,152.189
C01415=1103.065,421.375,402.370,-179.726,19.479,152.188
C01416=1103.060,421.128,402.411,-179.727,19.471,152.186
C01417=1103.053,420.881,402.450,-179.730,19.463,152.184
C01418=1103.048,420.635,402.490,-179.732,19.454,152.182
C01419=1103.042,420.387,402.530,-179.733,19.446,152.181
C01420=1103.036,420.141,402.570,-179.736,19.438,152.179
C01421=1103.030,419.895,402.610,-179.738,19.429,152.177
C01422=1103.025,419.648,402.650,-179.740,19.421,152.176
C01423=1103.019,419.400,402.690,-179.742,19.413,152.174
C01424=1103.013,419.155,402.729,-179.744,19.405,152.172
C01425=1103.008,418.907,402.769,-179.746,19.397,152.171
C01426=1103.001,418.661,402.809,-179.748,19.389,152.169
C01427=1102.996,418.414,402.849,-179.750,19.381,152.167
C01428=1102.990,418.167,402.889,-179.752,19.373,152.166
C01429=1102.984,417.920,402.929,-179.754,19.365,152.164
C01430=1102.979,417.674,402.968,-179.756,19.357,152.162
C01431=1102.972,417.427,403.008,-179.758,19.349,152.161
C01432=1102.968,417.181,403.048,-179.761,19.341,152.159
C01433=1102.961,416.933,403.087,-179.763,19.333,152.158
C01434=1102.955,416.686,403.126,-179.764,19.326,152.156
C01435=1102.950,416.441,403.166,-179.766,19.318,152.154
C01436=1102.944,416.193,403.206,-179.769,19.310,152.153
C01437=1102.938,415.946,403.246,-179.771,19.302,152.151
C01438=1102.933,415.700,403.285,-179.773,19.294,152.150
C01439=1102.927,415.452,403.324,-179.775,19.286,152.148
C01440=1102.921,415.207,403.364,-179.777,19.279,152.147
C01441=1102.915,414.959,403.403,-179.779,19.272,152.145
C01442=1102.909,414.712,403.443,-179.782,19.264,152.144
C01443=1102.903,414.466,403.482,-179.784,19.256,152.142
C01444=1102.897,414.219,403.521,-179.786,19.249,152.141
C01445=1102.892,413.972,403.560,-179.788,19.242,152.139
C01446=1102.886,413.725,403.600,-179.790,19.234,152.138
C01447=1102.880,413.478,403.639,-179.792,19.226,152.136
C01448=1102.874,413.232,403.678,-179.795,19.219,152.135
C01449=1102.868,412.984,403.718,-179.796,19.212,152.133
C01450=1102.863,412.738,403.757,-179.799,19.204,152.132
C01451=1102.856,412.491,403.796,-179.801,19.197,152.130
C01452=1102.851,412.244,403.835,-179.804,19.189,152.129
C01453=1102.845,411.997,403.875,-179.805,19.182,152.128
C01454=1102.839,411.751,403.914,-179.808,19.175,152.126
C01455=1102.833,411.504,403.953,-179.810,19.167,152.125
C01456=1102.828,411.289,403.987,-179.812,19.161,152.124
C01457=1102.824,411.076,404.021,-179.814,19.154,152.122
C01458=1102.819,410.862,404.054,-179.815,19.149,152.121
C01459=1102.814,410.647,404.089,-179.817,19.143,152.120
C01460=1102.809,410.433,404.123,-179.819,19.136,152.119
C01461=1102.804,410.218,404.157,-179.821,19.130,152.117
C01462=1102.799,410.005,404.191,-179.823,19.124,152.116
C01463=1102.794,409.791,404.224,-179.825,19.118,152.115
C01464=1102.788,409.544,404.264,-179.827,19.110,152.114
C01465=1102.783,409.297,404.302,-179.829,19.103,152.112
C01466=1102.777,409.050,404.341,-179.832,19.096,152.111
C01467=1102.771,408.803,404.380,-179.834,19.090,152.110
C01468=1102.765,408.556,404.418,-179.836,19.082,152.108
C01469=1102.759,408.309,404.458,-179.839,19.075,152.107
C01470=1102.754,408.063,404.497,-179.840,19.069,152.106
C01471=1102.749,407.816,404.535,-179.843,19.061,152.104
C01472=1102.743,407.569,404.574,-179.845,19.055,152.103
C01473=1102.737,407.322,404.612,-179.847,19.047,152.102
C01474=1102.731,407.075,404.652,-179.849,19.041,152.100
C01475=1102.726,406.828,404.690,-179.852,19.034,152.099
C01476=1102.720,406.581,404.729,-179.854,19.027,152.098
C01477=1102.714,406.334,404.767,-179.856,19.021,152.097
C01478=1102.708,406.087,404.806,-179.858,19.014,152.095
C01479=1102.702,405.840,404.845,-179.861,19.007,152.094
C01480=1102.697,405.593,404.884,-179.863,19.000,152.093
C01481=1102.691,405.346,404.922,-179.866,18.994,152.091
C01482=1102.685,405.099,404.961,-179.868,18.987,152.090
C01483=1102.680,404.852,405.000,-179.870,18.980,152.089
C01484=1102.674,404.605,405.037,-179.872,18.974,152.088
C01485=1102.668,404.358,405.077,-179.875,18.967,152.087
C01486=1102.662,404.112,405.114,-179.877,18.961,152.085
C01487=1102.657,403.864,405.153,-179.880,18.954,152.084
C01488=1102.651,403.617,405.192,-179.882,18.948,152.083
C01489=1102.645,403.371,405.230,-179.884,18.941,152.082
C01490=1102.639,403.124,405.268,-179.886,18.935,152.081
C01491=1102.633,402.877,405.307,-179.888,18.928,152.079
C01492=1102.628,402.630,405.346,-179.891,18.922,152.078
C01493=1102.622,402.383,405.383,-179.893,18.915,152.077
C01494=1102.616,402.135,405.422,-179.895,18.909,152.076
C01495=1102.610,401.888,405.460,-179.898,18.903,152.075
C01496=1102.604,401.642,405.499,-179.900,18.896,152.074
C01497=1102.599,401.395,405.537,-179.903,18.890,152.073
C01498=1102.593,401.147,405.575,-179.905,18.884,152.071
C01499=1102.587,400.901,405.613,-179.907,18.877,152.070
C01500=1102.582,400.654,405.651,-179.910,18.871,152.069
C01501=1102.576,400.407,405.689,-179.912,18.865,152.068
C01502=1102.571,400.160,405.728,-179.914,18.859,152.067
C01503=1102.564,399.912,405.766,-179.917,18.852,152.066
C01504=1102.559,399.665,405.804,-179.919,18.846,152.065
C01505=1102.553,399.419,405.842,-179.921,18.840,152.064
C01506=1102.547,399.172,405.880,-179.924,18.834,152.063
C01507=1102.541,398.924,405.918,-179.926,18.828,152.061
C01508=1102.535,398.677,405.956,-179.929,18.822,152.060
C01509=1102.530,398.431,405.994,-179.931,18.816,152.059
C01510=1102.524,398.184,406.032,-179.934,18.809,152.058
C01511=1102.519,397.937,406.070,-179.936,18.804,152.057
C01512=1102.513,397.723,406.103,-179.938,18.799,152.056
C01513=1102.509,397.508,406.135,-179.940,18.793,152.055
C01514=1102.503,397.294,406.168,-179.943,18.788,152.055
C01515=1102.498,397.080,406.202,-179.944,18.783,152.054
C01516=1102.493,396.866,406.234,-179.947,18.778,152.053
C01517=1102.489,396.652,406.267,-179.948,18.773,152.052
C01518=1102.483,396.438,406.300,-179.951,18.767,152.051
C01519=1102.479,396.223,406.333,-179.953,18.762,152.050
C01520=1102.473,395.976,406.370,-179.955,18.757,152.049
C01521=1102.467,395.730,406.408,-179.958,18.751,152.048
C01522=1102.461,395.483,406.446,-179.960,18.745,152.047
C01523=1102.456,395.235,406.484,-179.962,18.739,152.046
C01524=1102.450,394.989,406.521,-179.965,18.733,152.045
C01525=1102.444,394.742,406.559,-179.967,18.728,152.044
C01526=1102.438,394.494,406.597,-179.970,18.721,152.043
C01527=1102.432,394.247,406.634,-179.973,18.716,152.042
C01528=1102.426,394.000,406.672,-179.975,18.710,152.041
C01529=1102.421,393.753,406.709,-179.977,18.705,152.040
C01530=1102.416,393.506,406.747,-179.980,18.699,152.039
C01531=1102.410,393.259,406.785,-179.982,18.693,152.038
C01532=1102.404,393.012,406.822,-179.985,18.687,152.038
C01533=1102.398,392.765,406.860,-179.987,18.681,152.037
C01534=1102.392,392.518,406.897,-179.990,18.676,152.036
C01535=1102.387,392.271,406.935,-179.992,18.671,152.035
C01536=1102.381,392.024,406.973,-179.995,18.665,152.034
C01537=1102.375,391.777,407.010,-179.997,18.660,152.033
C01538=1102.369,391.530,407.047,-180.000,18.654,152.032
C01539=1102.364,391.283,407.084,179.998,18.649,152.031
C01540=1102.358,391.036,407.122,179.995,18.643,152.030
C01541=1102.352,390.789,407.159,179.992,18.637,152.029
C01542=1102.346,390.542,407.197,179.989,18.632,152.029
C01543=1102.340,390.295,407.233,179.987,18.627,152.028
C01544=1102.334,390.047,407.270,179.985,18.621,152.027
C01545=1102.328,389.801,407.308,179.982,18.616,152.026
C01546=1102.323,389.553,407.345,179.979,18.611,152.025
C01547=1102.317,389.307,407.383,179.977,18.605,152.024
C01548=1102.311,389.059,407.420,179.975,18.600,152.023
C01549=1102.306,388.812,407.457,179.972,18.595,152.023
C01550=1102.300,388.565,407.495,179.969,18.589,152.022
C01551=1102.293,388.318,407.531,179.966,18.584,152.021
C01552=1102.288,388.071,407.568,179.964,18.578,152.020
C01553=1102.282,387.823,407.605,179.961,18.573,152.019
C01554=1102.277,387.577,407.643,179.958,18.568,152.018
C01555=1102.271,387.330,407.680,179.956,18.563,152.018
C01556=1102.266,387.082,407.717,179.953,18.557,152.017
C01557=1102.259,386.835,407.753,179.951,18.552,152.016
C01558=1102.253,386.589,407.791,179.948,18.547,152.015
C01559=1102.248,386.341,407.828,179.946,18.541,152.014
C01560=1102.242,386.094,407.865,179.943,18.536,152.014
C01561=1102.237,385.847,407.902,179.940,18.531,152.013
C01562=1102.231,385.600,407.938,179.937,18.526,152.012
C01563=1102.225,385.353,407.975,179.935,18.521,152.011
C01564=1102.220,385.106,408.012,179.932,18.516,152.011
C01565=1102.214,384.858,408.049,179.930,18.511,152.010
C01566=1102.208,384.611,408.086,179.927,18.506,152.009
C01567=1102.203,384.364,408.122,179.924,18.501,152.008
C01568=1102.193,383.949,408.185,179.920,18.492,152.007
C01569=1102.183,383.533,408.247,179.915,18.483,152.006
C01570=1102.173,383.116,408.308,179.911,18.475,152.005
C01571=1102.164,382.701,408.370,179.907,18.467,152.003
C01572=1102.159,382.453,408.407,179.904,18.462,152.003
C01573=1102.152,382.206,408.443,179.901,18.457,152.002
C01574=1102.147,381.959,408.480,179.898,18.452,152.001
C01575=1102.142,381.712,408.517,179.896,18.447,152.001
C01576=1102.135,381.465,408.554,179.893,18.443,152.000
C01577=1102.130,381.217,408.590,179.890,18.437,151.999
C01578=1102.124,380.970,408.626,179.887,18.432,151.999
C01579=1102.118,380.723,408.663,179.885,18.428,151.998
C01580=1102.112,380.477,408.699,179.882,18.423,151.997
C01581=1102.107,380.229,408.737,179.879,18.418,151.997
C01582=1102.101,379.981,408.772,179.876,18.413,151.996
C01583=1102.095,379.734,408.809,179.874,18.409,151.995
C01584=1102.089,379.488,408.845,179.871,18.404,151.995
C01585=1102.083,379.240,408.881,179.869,18.399,151.994
C01586=1102.078,378.993,408.918,179.866,18.394,151.993
C01587=1102.072,378.746,408.954,179.863,18.390,151.993
C01588=1102.067,378.498,408.991,179.860,18.385,151.992
C01589=1102.060,378.251,409.027,179.857,18.380,151.991
C01590=1102.055,378.004,409.064,179.854,18.375,151.991
C01591=1102.049,377.757,409.099,179.852,18.371,151.990
C01592=1102.044,377.510,409.136,179.849,18.367,151.990
C01593=1102.038,377.262,409.172,179.846,18.362,151.989
C01594=1102.032,377.016,409.208,179.844,18.357,151.988
C01595=1102.027,376.768,409.245,179.841,18.352,151.988
C01596=1102.020,376.521,409.281,179.838,18.348,151.987
C01597=1102.016,376.273,409.317,179.836,18.343,151.986
C01598=1102.009,376.026,409.353,179.833,18.339,151.986
C01599=1102.004,375.779,409.389,179.830,18.334,151.985
C01600=1101.998,375.532,409.426,179.827,18.329,151.985
C01601=1101.992,375.284,409.462,179.824,18.325,151.984
C01602=1101.987,375.038,409.498,179.821,18.320,151.984
C01603=1101.981,374.790,409.534,179.819,18.316,151.983
C01604=1101.975,374.542,409.570,179.816,18.311,151.982
C01605=1101.970,374.296,409.606,179.813,18.307,151.982
C01606=1101.964,374.048,409.642,179.810,18.302,151.981
C01607=1101.959,373.801,409.677,179.807,18.298,151.981
C01608=1101.952,373.554,409.714,179.805,18.294,151.980
C01609=1101.946,373.306,409.750,179.802,18.289,151.980
C01610=1101.941,373.059,409.785,179.799,18.285,151.979
C01611=1101.935,372.812,409.821,179.796,18.281,151.979
C01612=1101.929,372.564,409.858,179.793,18.276,151.978
C01613=1101.924,372.317,409.893,179.790,18.272,151.978
C01614=1101.918,372.069,409.929,179.787,18.267,151.977
C01615=1101.912,371.823,409.965,179.784,18.263,151.977
C01616=1101.906,371.575,410.001,179.782,18.259,151.976
C01617=1101.900,371.328,410.036,179.779,18.255,151.976
C01618=1101.895,371.081,410.072,179.776,18.250,151.975
C01619=1101.889,370.833,410.107,179.773,18.246,151.975
C01620=1101.880,370.444,410.164,179.769,18.240,151.974
C01621=1101.871,370.055,410.221,179.765,18.233,151.973
C01622=1101.862,369.667,410.276,179.760,18.226,151.972
C01623=1101.854,369.277,410.332,179.755,18.220,151.971
C01624=1101.848,369.029,410.368,179.752,18.215,151.971
C01625=1101.842,368.782,410.403,179.749,18.211,151.971
C01626=1101.836,368.535,410.439,179.747,18.207,151.970
C01627=1101.831,368.288,410.474,179.744,18.203,151.970
C01628=1101.825,368.040,410.510,179.741,18.199,151.969
C01629=1101.819,367.793,410.545,179.738,18.195,151.969
C01630=1101.813,367.545,410.581,179.735,18.191,151.968
C01631=1101.808,367.298,410.616,179.732,18.186,151.968
C01632=1101.802,367.051,410.652,179.729,18.182,151.967
C01633=1101.796,366.804,410.688,179.726,18.178,151.967
C01634=1101.791,366.557,410.723,179.723,18.174,151.966
C01635=1101.785,366.308,410.758,179.720,18.170,151.966
C01636=1101.780,366.062,410.793,179.718,18.166,151.966
C01637=1101.774,365.814,410.829,179.714,18.162,151.965
C01638=1101.768,365.567,410.864,179.711,18.158,151.965
C01639=1101.762,365.319,410.900,179.709,18.154,151.964
C01640=1101.757,365.072,410.935,179.706,18.150,151.964
C01641=1101.750,364.824,410.970,179.703,18.146,151.964
C01642=1101.745,364.577,411.005,179.700,18.142,151.963
C01643=1101.739,364.330,411.041,179.697,18.138,151.963
C01644=1101.734,364.082,411.076,179.694,18.134,151.962
C01645=1101.728,363.835,411.111,179.691,18.130,151.962
C01646=1101.722,363.588,411.146,179.688,18.126,151.961
C01647=1101.716,363.340,411.181,179.685,18.122,151.961
C01648=1101.710,363.092,411.216,179.682,18.119,151.961
C01649=1101.705,362.845,411.251,179.680,18.115,151.960
C01650=1101.700,362.598,411.286,179.676,18.111,151.960
C01651=1101.693,362.350,411.322,179.673,18.107,151.960
C01652=1101.688,362.103,411.356,179.670,18.103,151.959
C01653=1101.682,361.855,411.392,179.667,18.099,151.959
C01654=1101.677,361.608,411.427,179.665,18.096,151.959
C01655=1101.671,361.361,411.461,179.661,18.092,151.958
C01656=1101.665,361.113,411.496,179.658,18.088,151.958
C01657=1101.659,360.866,411.532,179.656,18.084,151.957
C01658=1101.654,360.618,411.566,179.652,18.080,151.957
C01659=1101.648,360.371,411.602,179.650,18.077,151.957
C01660=1101.642,360.123,411.636,179.646,18.073,151.956
C01661=1101.636,359.875,411.672,179.643,18.069,151.956
C01662=1101.631,359.628,411.706,179.641,18.065,151.956
C01663=1101.625,359.381,411.741,179.637,18.061,151.955
C01664=1101.619,359.133,411.776,179.635,18.058,151.955
C01665=1101.614,358.886,411.810,179.631,18.054,151.955
C01666=1101.608,358.638,411.845,179.628,18.051,151.955
C01667=1101.602,358.391,411.880,179.625,18.047,151.954
C01668=1101.597,358.143,411.915,179.623,18.043,151.954
C01669=1101.591,357.896,411.949,179.619,18.040,151.954
C01670=1101.585,357.648,411.985,179.617,18.036,151.953
C01671=1101.579,357.401,412.019,179.613,18.032,151.953
C01672=1101.570,357.026,412.071,179.608,18.027,151.953
C01673=1101.562,356.653,412.124,179.604,18.021,151.952
C01674=1101.553,356.278,412.176,179.599,18.015,151.952
C01675=1101.545,355.904,412.228,179.595,18.011,151.951
C01676=1101.539,355.656,412.262,179.592,18.007,151.951
C01677=1101.533,355.409,412.298,179.589,18.003,151.951
C01678=1101.527,355.162,412.332,179.586,18.000,151.950
C01679=1101.522,354.915,412.366,179.583,17.997,151.950
C01680=1101.516,354.667,412.401,179.580,17.993,151.950
C01681=1101.511,354.419,412.435,179.577,17.990,151.950
C01682=1101.505,354.172,412.469,179.573,17.986,151.949
C01683=1101.500,353.924,412.504,179.571,17.982,151.949
C01684=1101.494,353.677,412.538,179.567,17.979,151.949
C01685=1101.488,353.428,412.573,179.565,17.975,151.948
C01686=1101.482,353.181,412.607,179.561,17.972,151.948
C01687=1101.476,352.934,412.641,179.558,17.969,151.948
C01688=1101.471,352.686,412.676,179.555,17.965,151.948
C01689=1101.465,352.438,412.710,179.552,17.962,151.948
C01690=1101.459,352.191,412.744,179.549,17.958,151.947
C01691=1101.454,351.943,412.779,179.546,17.955,151.947
C01692=1101.448,351.696,412.813,179.542,17.951,151.947
C01693=1101.442,351.449,412.847,179.540,17.948,151.947
C01694=1101.437,351.200,412.881,179.537,17.945,151.946
C01695=1101.431,350.953,412.916,179.533,17.941,151.946
C01696=1101.425,350.705,412.950,179.531,17.938,151.946
C01697=1101.419,350.458,412.984,179.527,17.935,151.946
C01698=1101.414,350.211,413.018,179.525,17.931,151.946
C01699=1101.408,349.963,413.052,179.521,17.928,151.945
C01700=1101.402,349.715,413.086,179.518,17.925,151.945
C01701=1101.396,349.467,413.120,179.515,17.922,151.945
C01702=1101.391,349.220,413.155,179.512,17.918,151.945
C01703=1101.385,348.972,413.189,179.509,17.915,151.945
C01704=1101.379,348.725,413.222,179.506,17.911,151.944
C01705=1101.374,348.477,413.256,179.503,17.908,151.944
C01706=1101.368,348.230,413.291,179.499,17.905,151.944
C01707=1101.363,347.982,413.324,179.496,17.902,151.944
C01708=1101.356,347.734,413.359,179.493,17.899,151.944
C01709=1101.351,347.487,413.393,179.490,17.895,151.943
C01710=1101.345,347.239,413.426,179.487,17.892,151.943
C01711=1101.339,346.991,413.460,179.483,17.888,151.943
C01712=1101.334,346.743,413.494,179.481,17.886,151.943
C01713=1101.329,346.496,413.528,179.478,17.882,151.943
C01714=1101.323,346.249,413.562,179.474,17.879,151.943
C01715=1101.317,346.001,413.595,179.471,17.876,151.942
C01716=1101.311,345.753,413.629,179.469,17.873,151.942
C01717=1101.306,345.505,413.663,179.465,17.869,151.942
C01718=1101.300,345.258,413.697,179.462,17.866,151.942
C01719=1101.294,345.010,413.730,179.459,17.863,151.942
C01720=1101.288,344.763,413.764,179.456,17.860,151.942
C01721=1101.283,344.515,413.798,179.453,17.857,151.942
C01722=1101.277,344.266,413.831,179.449,17.854,151.941
C01723=1101.271,344.019,413.865,179.446,17.851,151.941
C01724=1101.263,343.647,413.915,179.442,17.846,151.941
C01725=1101.254,343.276,413.966,179.437,17.842,151.941
C01726=1101.246,342.904,414.016,179.432,17.837,151.941
C01727=1101.237,342.531,414.067,179.427,17.833,151.941
C01728=1101.231,342.284,414.100,179.424,17.830,151.940
C01729=1101.225,342.036,414.134,179.421,17.826,151.940
C01730=1101.220,341.789,414.167,179.418,17.823,151.940
C01731=1101.214,341.541,414.201,179.415,17.821,151.940
C01732=1101.208,341.293,414.235,179.411,17.817,151.940
C01733=1101.203,341.045,414.268,179.408,17.814,151.940
C01734=1101.197,340.798,414.301,179.405,17.811,151.940
C01735=1101.191,340.550,414.335,179.402,17.808,151.940
C01736=1101.186,340.302,414.369,179.399,17.806,151.940
C01737=1101.181,340.055,414.402,179.396,17.803,151.939
C01738=1101.174,339.808,414.434,179.393,17.800,151.939
C01739=1101.169,339.560,414.468,179.389,17.796,151.939
C01740=1101.163,339.312,414.501,179.386,17.794,151.939
C01741=1101.158,339.064,414.534,179.383,17.791,151.939
C01742=1101.152,338.817,414.568,179.379,17.788,151.939
C01743=1101.146,338.569,414.602,179.376,17.785,151.939
C01744=1101.140,338.321,414.634,179.374,17.782,151.939
C01745=1101.135,338.073,414.668,179.370,17.779,151.939
C01746=1101.129,337.825,414.701,179.367,17.776,151.939
C01747=1101.123,337.577,414.734,179.364,17.773,151.939
C01748=1101.117,337.330,414.767,179.361,17.771,151.939
C01749=1101.112,337.082,414.801,179.358,17.768,151.938
C01750=1101.106,336.834,414.834,179.354,17.765,151.938
C01751=1101.100,336.587,414.866,179.351,17.762,151.938
C01752=1101.095,336.339,414.900,179.348,17.760,151.938
C01753=1101.089,336.091,414.933,179.345,17.757,151.938
C01754=1101.084,335.843,414.966,179.341,17.753,151.938
C01755=1101.077,335.596,414.999,179.338,17.751,151.938
C01756=1101.072,335.347,415.032,179.335,17.748,151.938
C01757=1101.066,335.100,415.064,179.332,17.745,151.938
C01758=1101.060,334.852,415.098,179.328,17.742,151.938
C01759=1101.055,334.605,415.131,179.325,17.740,151.938
C01760=1101.049,334.357,415.163,179.322,17.737,151.938
C01761=1101.043,334.109,415.197,179.319,17.734,151.938
C01762=1101.038,333.861,415.230,179.315,17.731,151.938
C01763=1101.032,333.613,415.262,179.312,17.728,151.938
C01764=1101.027,333.366,415.295,179.309,17.726,151.938
C01765=1101.021,333.118,415.328,179.306,17.723,151.938
C01766=1101.015,332.870,415.361,179.303,17.721,151.938
C01767=1101.010,332.622,415.394,179.299,17.717,151.938
C01768=1101.004,332.374,415.427,179.296,17.715,151.938
C01769=1100.999,332.127,415.460,179.293,17.712,151.938
C01770=1100.993,331.879,415.492,179.290,17.710,151.938
C01771=1100.987,331.631,415.525,179.287,17.707,151.938
C01772=1100.981,331.383,415.558,179.284,17.705,151.938
C01773=1100.975,331.135,415.590,179.280,17.702,151.938
C01774=1100.969,330.887,415.623,179.277,17.699,151.938
C01775=1100.964,330.640,415.655,179.274,17.697,151.938
C01776=1100.955,330.262,415.706,179.269,17.693,151.938
C01777=1100.946,329.884,415.755,179.263,17.689,151.938
C01778=1100.937,329.506,415.804,179.259,17.685,151.938
C01779=1100.929,329.128,415.854,179.254,17.681,151.938
C01780=1100.923,328.880,415.887,179.251,17.679,151.938
C01781=1100.917,328.632,415.919,179.247,17.676,151.938
C01782=1100.911,328.384,415.952,179.244,17.673,151.938
C01783=1100.906,328.137,415.984,179.241,17.671,151.938
C01784=1100.899,327.889,416.017,179.237,17.668,151.938
C01785=1100.893,327.641,416.049,179.234,17.666,151.938
C01786=1100.888,327.392,416.081,179.231,17.663,151.938
C01787=1100.882,327.146,416.114,179.228,17.661,151.938
C01788=1100.876,326.897,416.146,179.224,17.658,151.938
C01789=1100.871,326.649,416.179,179.221,17.655,151.938
C01790=1100.865,326.402,416.211,179.218,17.653,151.938
C01791=1100.859,326.154,416.243,179.215,17.651,151.938
C01792=1100.853,325.906,416.275,179.211,17.648,151.938
C01793=1100.848,325.658,416.308,179.208,17.646,151.938
C01794=1100.843,325.410,416.340,179.205,17.643,151.938
C01795=1100.836,325.162,416.373,179.202,17.641,151.938
C01796=1100.831,324.915,416.404,179.198,17.639,151.939
C01797=1100.825,324.667,416.436,179.194,17.636,151.939
C01798=1100.820,324.418,416.469,179.191,17.633,151.939
C01799=1100.814,324.171,416.501,179.188,17.631,151.939
C01800=1100.808,323.923,416.533,179.185,17.628,151.939
